LIN {X 0,Y 509.862,Z 318.469,A -85,B 0,C 180,E1 -5560.681,E2 -5560.681} C_VEL
LIN {X 0,Y 509.875,Z 318.471,A -85,B 0,C 180,E1 -5563.174,E2 -5563.174} C_VEL
LIN {X 0,Y 509.873,Z 318.475,A -85,B 0,C 180,E1 -5565.634,E2 -5565.634} C_VEL
LIN {X 0,Y 509.913,Z 318.465,A -85,B 0,C 180,E1 -5568.874,E2 -5568.874} C_VEL
LIN {X 0,Y 509.951,Z 318.459,A -85,B 0,C 180,E1 -5572.078,E2 -5572.078} C_VEL
LIN {X 0,Y 509.98,Z 318.455,A -85,B 0,C 180,E1 -5574.464,E2 -5574.464} C_VEL
LIN {X 0,Y 510.056,Z 318.449,A -85,B 0,C 180,E1 -5577.63,E2 -5577.63} C_VEL
LIN {X 0,Y 510.062,Z 318.448,A -85,B 0,C 180,E1 -5580.789,E2 -5580.789} C_VEL
LIN {X 0,Y 509.954,Z 318.466,A -85,B 0,C 180,E1 -5583.16,E2 -5583.16} C_VEL
LIN {X 0,Y 509.953,Z 318.459,A -85,B 0,C 180,E1 -5586.329,E2 -5586.329} C_VEL
LIN {X 0,Y 509.913,Z 318.468,A -85,B 0,C 180,E1 -5588.72,E2 -5588.72} C_VEL
LIN {X 0,Y 509.903,Z 318.464,A -85,B 0,C 180,E1 -5591.931,E2 -5591.931} C_VEL
LIN {X 0,Y 509.892,Z 318.469,A -85,B 0,C 180,E1 -5595.241,E2 -5595.241} C_VEL
LIN {X 0,Y 509.887,Z 318.467,A -85,B 0,C 180,E1 -5598.001,E2 -5598.001} C_VEL
LIN {X 0,Y 509.848,Z 318.475,A -85,B 0,C 180,E1 -5601.001,E2 -5601.001} C_VEL
LIN {X 0,Y 509.862,Z 318.476,A -85,B 0,C 180,E1 -5604.426,E2 -5604.426} C_VEL
LIN {X 0,Y 509.882,Z 318.469,A -85,B 0,C 180,E1 -5607.055,E2 -5607.055} C_VEL
LIN {X 0,Y 509.854,Z 318.471,A -85,B 0,C 180,E1 -5609.751,E2 -5609.751} C_VEL
LIN {X 0,Y 509.874,Z 318.471,A -85,B 0,C 180,E1 -5612.774,E2 -5612.774} C_VEL
LIN {X 0,Y 509.836,Z 318.473,A -85,B 0,C 180,E1 -5615.58,E2 -5615.58} C_VEL
LIN {X 0,Y 509.849,Z 318.479,A -85,B 0,C 180,E1 -5618.337,E2 -5618.337} C_VEL
LIN {X 0,Y 509.862,Z 318.47,A -85,B 0,C 180,E1 -5621.424,E2 -5621.424} C_VEL
LIN {X 0,Y 509.853,Z 318.472,A -85,B 0,C 180,E1 -5624.668,E2 -5624.668} C_VEL
LIN {X 0,Y 509.858,Z 318.478,A -85,B 0,C 180,E1 -5628.102,E2 -5628.102} C_VEL
LIN {X 0,Y 509.857,Z 318.471,A -85,B 0,C 180,E1 -5630.649,E2 -5630.649} C_VEL
LIN {X 0,Y 509.827,Z 318.478,A -85,B 0,C 180,E1 -5633.723,E2 -5633.723} C_VEL
LIN {X 0,Y 509.159,Z 318.56,A -85,B 0,C 180,E1 -5634.382,E2 -5634.382} C_VEL
LIN {X 0,Y 506.343,Z 318.911,A -85,B 0,C 180,E1 -5635.454,E2 -5635.454} C_VEL
LIN {X 0,Y 503.953,Z 319.208,A -85,B 0,C 180,E1 -5636.318,E2 -5636.318} C_VEL
LIN {X 0,Y 502.905,Z 319.336,A -85,B 0,C 180,E1 -5636.984,E2 -5636.984} C_VEL
LIN {X 0,Y 502.807,Z 319.349,A -85,B 0,C 180,E1 -5637.21,E2 -5637.21} C_VEL
LIN {X 0,Y 502.811,Z 319.352,A -85,B 0,C 180,E1 -5640.065,E2 -5640.065} C_VEL
LIN {X 0,Y 502.832,Z 319.345,A -85,B 0,C 180,E1 -5642.533,E2 -5642.533} C_VEL
LIN {X 0,Y 502.823,Z 319.351,A -85,B 0,C 180,E1 -5645.299,E2 -5645.299} C_VEL
LIN {X 0,Y 502.776,Z 319.357,A -85,B 0,C 180,E1 -5647.826,E2 -5647.826} C_VEL
LIN {X 0,Y 502.822,Z 319.346,A -85,B 0,C 180,E1 -5650.4,E2 -5650.4} C_VEL
LIN {X 0,Y 502.831,Z 319.35,A -85,B 0,C 180,E1 -5652.932,E2 -5652.932} C_VEL
LIN {X 0,Y 502.848,Z 319.352,A -85,B 0,C 180,E1 -5655.429,E2 -5655.429} C_VEL
LIN {X 0,Y 502.874,Z 319.343,A -85,B 0,C 180,E1 -5658.717,E2 -5658.717} C_VEL
LIN {X 0,Y 502.899,Z 319.34,A -85,B 0,C 180,E1 -5661.967,E2 -5661.967} C_VEL
LIN {X 0,Y 502.939,Z 319.335,A -85,B 0,C 180,E1 -5664.387,E2 -5664.387} C_VEL
LIN {X 0,Y 503.023,Z 319.325,A -85,B 0,C 180,E1 -5667.598,E2 -5667.598} C_VEL
LIN {X 0,Y 503.025,Z 319.324,A -85,B 0,C 180,E1 -5670,E2 -5670} C_VEL
LIN {X 0,Y 503.023,Z 319.325,A -85,B 0,C 180,E1 -5672.402,E2 -5672.402} C_VEL
LIN {X 0,Y 502.939,Z 319.335,A -85,B 0,C 180,E1 -5675.613,E2 -5675.613} C_VEL
LIN {X 0,Y 502.899,Z 319.34,A -85,B 0,C 180,E1 -5678.033,E2 -5678.033} C_VEL
LIN {X 0,Y 502.874,Z 319.343,A -85,B 0,C 180,E1 -5681.283,E2 -5681.283} C_VEL
LIN {X 0,Y 502.848,Z 319.352,A -85,B 0,C 180,E1 -5684.571,E2 -5684.571} C_VEL
LIN {X 0,Y 502.859,Z 319.345,A -85,B 0,C 180,E1 -5687.907,E2 -5687.907} C_VEL
LIN {X 0,Y 502.825,Z 319.354,A -85,B 0,C 180,E1 -5690.536,E2 -5690.536} C_VEL
LIN {X 0,Y 502.788,Z 319.352,A -85,B 0,C 180,E1 -5693.041,E2 -5693.041} C_VEL
LIN {X 0,Y 502.838,Z 319.345,A -85,B 0,C 180,E1 -5695.676,E2 -5695.676} C_VEL
LIN {X 0,Y 502.837,Z 319.353,A -85,B 0,C 180,E1 -5698.373,E2 -5698.373} C_VEL
LIN {X 0,Y 502.793,Z 319.351,A -85,B 0,C 180,E1 -5701.5,E2 -5701.5} C_VEL
LIN {X 0,Y 502.801,Z 319.354,A -85,B 0,C 180,E1 -5704.444,E2 -5704.444} C_VEL
LIN {X 0,Y 502.777,Z 319.352,A -85,B 0,C 180,E1 -5707.178,E2 -5707.178} C_VEL
LIN {X 0,Y 502.818,Z 319.356,A -85,B 0,C 180,E1 -5710.012,E2 -5710.012} C_VEL
LIN {X 0,Y 502.77,Z 319.354,A -85,B 0,C 180,E1 -5713.231,E2 -5713.231} C_VEL
LIN {X 0,Y 502.787,Z 319.356,A -85,B 0,C 180,E1 -5715.662,E2 -5715.662} C_VEL
LIN {X 0,Y 502.832,Z 319.354,A -85,B 0,C 180,E1 -5717.865,E2 -5717.865} C_VEL
LIN {X 0,Y 502.807,Z 319.349,A -85,B 0,C 180,E1 -5721.025,E2 -5721.025} C_VEL
LIN {X 0,Y 502.771,Z 319.355,A -85,B 0,C 180,E1 -5724.169,E2 -5724.169} C_VEL
LIN {X 0,Y 502.83,Z 319.347,A -85,B 0,C 180,E1 -5726.994,E2 -5726.994} C_VEL
LIN {X 0,Y 502.812,Z 319.35,A -85,B 0,C 180,E1 -5730.065,E2 -5730.065} C_VEL
LIN {X 0,Y 502.831,Z 319.345,A -85,B 0,C 180,E1 -5732.534,E2 -5732.534} C_VEL
LIN {X 0,Y 502.824,Z 319.353,A -85,B 0,C 180,E1 -5735.299,E2 -5735.299} C_VEL
LIN {X 0,Y 502.778,Z 319.354,A -85,B 0,C 180,E1 -5737.827,E2 -5737.827} C_VEL
LIN {X 0,Y 502.823,Z 319.346,A -85,B 0,C 180,E1 -5740.401,E2 -5740.401} C_VEL
LIN {X 0,Y 502.832,Z 319.35,A -85,B 0,C 180,E1 -5742.932,E2 -5742.932} C_VEL
LIN {X 0,Y 502.843,Z 319.349,A -85,B 0,C 180,E1 -5745.43,E2 -5745.43} C_VEL
LIN {X 0,Y 502.876,Z 319.343,A -85,B 0,C 180,E1 -5748.717,E2 -5748.717} C_VEL
LIN {X 0,Y 502.9,Z 319.337,A -85,B 0,C 180,E1 -5751.967,E2 -5751.967} C_VEL
LIN {X 0,Y 502.933,Z 319.334,A -85,B 0,C 180,E1 -5754.387,E2 -5754.387} C_VEL
LIN {X 0,Y 503.024,Z 319.322,A -85,B 0,C 180,E1 -5757.598,E2 -5757.598} C_VEL
LIN {X 0,Y 503.034,Z 319.329,A -85,B 0,C 180,E1 -5760.801,E2 -5760.801} C_VEL
LIN {X 0,Y 502.896,Z 319.34,A -85,B 0,C 180,E1 -5763.205,E2 -5763.205} C_VEL
LIN {X 0,Y 502.906,Z 319.341,A -85,B 0,C 180,E1 -5766.419,E2 -5766.419} C_VEL
LIN {X 0,Y 502.874,Z 319.345,A -85,B 0,C 180,E1 -5768.844,E2 -5768.844} C_VEL
LIN {X 0,Y 502.846,Z 319.346,A -85,B 0,C 180,E1 -5772.102,E2 -5772.102} C_VEL
LIN {X 0,Y 502.849,Z 319.343,A -85,B 0,C 180,E1 -5775.4,E2 -5775.4} C_VEL
LIN {X 0,Y 502.826,Z 319.349,A -85,B 0,C 180,E1 -5778.752,E2 -5778.752} C_VEL
LIN {X 0,Y 502.783,Z 319.351,A -85,B 0,C 180,E1 -5781.312,E2 -5781.312} C_VEL
LIN {X 0,Y 502.776,Z 319.356,A -85,B 0,C 180,E1 -5783.915,E2 -5783.915} C_VEL
LIN {X 0,Y 502.865,Z 319.344,A -85,B 0,C 180,E1 -5786.566,E2 -5786.566} C_VEL
LIN {X 0,Y 502.824,Z 319.346,A -85,B 0,C 180,E1 -5789.288,E2 -5789.288} C_VEL
LIN {X 0,Y 502.784,Z 319.36,A -85,B 0,C 180,E1 -5792.085,E2 -5792.085} C_VEL
LIN {X 0,Y 502.799,Z 319.349,A -85,B 0,C 180,E1 -5794.966,E2 -5794.966} C_VEL
LIN {X 0,Y 502.794,Z 319.359,A -85,B 0,C 180,E1 -5797.954,E2 -5797.954} C_VEL
LIN {X 0,Y 502.821,Z 319.352,A -85,B 0,C 180,E1 -5801.066,E2 -5801.066} C_VEL
LIN {X 0,Y 502.792,Z 319.531,A -85,B 0,C 180,E1 -5803.377,E2 -5803.377} C_VEL
LIN {X 0,Y 503.366,Z 323.551,A -85,B 0,C 180,E1 -5806.555,E2 -5806.555} C_VEL
LIN {X 0,Y 503.464,Z 326.838,A -85,B 0,C 180,E1 -5808.921,E2 -5808.921} C_VEL
LIN {X 0,Y 503.339,Z 331.622,A -85,B 0,C 180,E1 -5812.095,E2 -5812.095} C_VEL
LIN {X 0,Y 503.119,Z 336.421,A -85,B 0,C 180,E1 -5815.06,E2 -5815.06} C_VEL
LIN {X 0,Y 502.955,Z 341.324,A -85,B 0,C 180,E1 -5817.928,E2 -5817.928} C_VEL
LIN {X 0,Y 502.767,Z 346.348,A -85,B 0,C 180,E1 -5820.709,E2 -5820.709} C_VEL
LIN {X 0,Y 502.617,Z 351.579,A -85,B 0,C 180,E1 -5823.496,E2 -5823.496} C_VEL
LIN {X 0,Y 502.426,Z 356.59,A -85,B 0,C 180,E1 -5826.068,E2 -5826.068} C_VEL
LIN {X 0,Y 502.342,Z 361.823,A -85,B 0,C 180,E1 -5828.669,E2 -5828.669} C_VEL
LIN {X 0,Y 502.248,Z 367.111,A -85,B 0,C 180,E1 -5831.226,E2 -5831.226} C_VEL
LIN {X 0,Y 502.175,Z 372.422,A -85,B 0,C 180,E1 -5833.746,E2 -5833.746} C_VEL
LIN {X 0,Y 502.176,Z 376.661,A -85,B 0,C 180,E1 -5835.72,E2 -5835.72} C_VEL
LIN {X 0,Y 504.336,Z 390.065,A -85,B 0,C 180,E1 -5836.133,E2 -5836.133} C_VEL
LIN {X 0,Y 504.45,Z 397.294,A -85,B 0,C 180,E1 -5836.402,E2 -5836.402} C_VEL
LIN {X 0,Y 504.208,Z 406.373,A -85,B 0,C 180,E1 -5836.806,E2 -5836.806} C_VEL
LIN {X 0,Y 503.872,Z 416.43,A -85,B 0,C 180,E1 -5837.368,E2 -5837.368} C_VEL
LIN {X 0,Y 503.598,Z 424.509,A -85,B 0,C 180,E1 -5837.917,E2 -5837.917} C_VEL
LIN {X 0,Y 503.364,Z 433.242,A -85,B 0,C 180,E1 -5838.626,E2 -5838.626} C_VEL
LIN {X 0,Y 503.096,Z 440.64,A -85,B 0,C 180,E1 -5839.333,E2 -5839.333} C_VEL
LIN {X 0,Y 502.873,Z 447.862,A -85,B 0,C 180,E1 -5840.142,E2 -5840.142} C_VEL
LIN {X 0,Y 502.658,Z 454.064,A -85,B 0,C 180,E1 -5840.95,E2 -5840.95} C_VEL
LIN {X 0,Y 502.487,Z 460.603,A -85,B 0,C 180,E1 -5841.96,E2 -5841.96} C_VEL
LIN {X 0,Y 502.332,Z 466.157,A -85,B 0,C 180,E1 -5842.989,E2 -5842.989} C_VEL
LIN {X 0,Y 502.233,Z 470.593,A -85,B 0,C 180,E1 -5843.976,E2 -5843.976} C_VEL
LIN {X 0,Y 502.115,Z 474.913,A -85,B 0,C 180,E1 -5845.183,E2 -5845.183} C_VEL
LIN {X 0,Y 502.14,Z 477.278,A -85,B 0,C 180,E1 -5845.987,E2 -5845.987} C_VEL
LIN {X 0,Y 502.121,Z 479.073,A -85,B 0,C 180,E1 -5846.791,E2 -5846.791} C_VEL
LIN {X 0,Y 502.037,Z 481.512,A -85,B 0,C 180,E1 -5848.396,E2 -5848.396} C_VEL
LIN {X 0,Y 501.99,Z 482.097,A -85,B 0,C 180,E1 -5849.198,E2 -5849.198} C_VEL
LIN {X 0,Y 501.99,Z 482.097,A -85,B 0,C 180,E1 -5850.802,E2 -5850.802} C_VEL
LIN {X 0,Y 502.037,Z 481.512,A -85,B 0,C 180,E1 -5851.604,E2 -5851.604} C_VEL
LIN {X 0,Y 502.121,Z 479.073,A -85,B 0,C 180,E1 -5853.209,E2 -5853.209} C_VEL
LIN {X 0,Y 502.107,Z 476.128,A -85,B 0,C 180,E1 -5854.415,E2 -5854.415} C_VEL
LIN {X 0,Y 502.217,Z 472.146,A -85,B 0,C 180,E1 -5855.622,E2 -5855.622} C_VEL
LIN {X 0,Y 502.277,Z 467.21,A -85,B 0,C 180,E1 -5856.79,E2 -5856.79} C_VEL
LIN {X 0,Y 502.418,Z 461.757,A -85,B 0,C 180,E1 -5857.839,E2 -5857.839} C_VEL
LIN {X 0,Y 502.611,Z 455.441,A -85,B 0,C 180,E1 -5858.848,E2 -5858.848} C_VEL
LIN {X 0,Y 502.826,Z 449.489,A -85,B 0,C 180,E1 -5859.655,E2 -5859.655} C_VEL
LIN {X 0,Y 503.01,Z 442.559,A -85,B 0,C 180,E1 -5860.465,E2 -5860.465} C_VEL
LIN {X 0,Y 503.324,Z 434.377,A -85,B 0,C 180,E1 -5861.273,E2 -5861.273} C_VEL
LIN {X 0,Y 503.624,Z 425.863,A -85,B 0,C 180,E1 -5861.98,E2 -5861.98} C_VEL
LIN {X 0,Y 503.807,Z 417.91,A -85,B 0,C 180,E1 -5862.541,E2 -5862.541} C_VEL
LIN {X 0,Y 504.092,Z 408.386,A -85,B 0,C 180,E1 -5863.094,E2 -5863.094} C_VEL
LIN {X 0,Y 504.404,Z 398.582,A -85,B 0,C 180,E1 -5863.548,E2 -5863.548} C_VEL
LIN {X 0,Y 504.443,Z 390.833,A -85,B 0,C 180,E1 -5863.842,E2 -5863.842} C_VEL
LIN {X 0,Y 502.465,Z 378.896,A -85,B 0,C 180,E1 -5864.217,E2 -5864.217} C_VEL
LIN {X 0,Y 502.167,Z 376.661,A -85,B 0,C 180,E1 -5864.28,E2 -5864.28} C_VEL
LIN {X 0,Y 502.212,Z 370.632,A -85,B 0,C 180,E1 -5867.09,E2 -5867.09} C_VEL
LIN {X 0,Y 502.34,Z 363.567,A -85,B 0,C 180,E1 -5870.473,E2 -5870.473} C_VEL
LIN {X 0,Y 502.406,Z 358.325,A -85,B 0,C 180,E1 -5873.059,E2 -5873.059} C_VEL
LIN {X 0,Y 502.533,Z 353.134,A -85,B 0,C 180,E1 -5875.692,E2 -5875.692} C_VEL
LIN {X 0,Y 502.692,Z 347.991,A -85,B 0,C 180,E1 -5878.382,E2 -5878.382} C_VEL
LIN {X 0,Y 502.89,Z 342.977,A -85,B 0,C 180,E1 -5881.137,E2 -5881.137} C_VEL
LIN {X 0,Y 503.066,Z 338.021,A -85,B 0,C 180,E1 -5883.974,E2 -5883.974} C_VEL
LIN {X 0,Y 503.247,Z 333.191,A -85,B 0,C 180,E1 -5886.906,E2 -5886.906} C_VEL
LIN {X 0,Y 503.406,Z 328.47,A -85,B 0,C 180,E1 -5889.956,E2 -5889.956} C_VEL
LIN {X 0,Y 503.471,Z 325.105,A -85,B 0,C 180,E1 -5892.282,E2 -5892.282} C_VEL
LIN {X 0,Y 503.174,Z 322.074,A -85,B 0,C 180,E1 -5894.574,E2 -5894.574} C_VEL
LIN {X 0,Y 502.774,Z 319.359,A -85,B 0,C 180,E1 -5896.768,E2 -5896.768} C_VEL
LIN {X 0,Y 502.819,Z 319.352,A -85,B 0,C 180,E1 -5899.005,E2 -5899.005} C_VEL
LIN {X 0,Y 502.794,Z 319.359,A -85,B 0,C 180,E1 -5902.046,E2 -5902.046} C_VEL
LIN {X 0,Y 502.799,Z 319.352,A -85,B 0,C 180,E1 -5905.034,E2 -5905.034} C_VEL
LIN {X 0,Y 502.784,Z 319.36,A -85,B 0,C 180,E1 -5907.915,E2 -5907.915} C_VEL
LIN {X 0,Y 502.824,Z 319.346,A -85,B 0,C 180,E1 -5910.712,E2 -5910.712} C_VEL
LIN {X 0,Y 502.863,Z 319.345,A -85,B 0,C 180,E1 -5913.439,E2 -5913.439} C_VEL
LIN {X 0,Y 502.776,Z 319.356,A -85,B 0,C 180,E1 -5916.085,E2 -5916.085} C_VEL
LIN {X 0,Y 502.783,Z 319.351,A -85,B 0,C 180,E1 -5918.688,E2 -5918.688} C_VEL
LIN {X 0,Y 502.826,Z 319.349,A -85,B 0,C 180,E1 -5921.248,E2 -5921.248} C_VEL
LIN {X 0,Y 502.849,Z 319.343,A -85,B 0,C 180,E1 -5924.6,E2 -5924.6} C_VEL
LIN {X 0,Y 502.876,Z 319.341,A -85,B 0,C 180,E1 -5928.039,E2 -5928.039} C_VEL
LIN {X 0,Y 502.874,Z 319.345,A -85,B 0,C 180,E1 -5931.156,E2 -5931.156} C_VEL
LIN {X 0,Y 502.906,Z 319.341,A -85,B 0,C 180,E1 -5933.581,E2 -5933.581} C_VEL
LIN {X 0,Y 502.896,Z 319.34,A -85,B 0,C 180,E1 -5936.795,E2 -5936.795} C_VEL
LIN {X 0,Y 503.034,Z 319.329,A -85,B 0,C 180,E1 -5939.199,E2 -5939.199} C_VEL
LIN {X 0,Y 503.024,Z 319.322,A -85,B 0,C 180,E1 -5942.402,E2 -5942.402} C_VEL
LIN {X 0,Y 502.933,Z 319.334,A -85,B 0,C 180,E1 -5945.613,E2 -5945.613} C_VEL
LIN {X 0,Y 502.9,Z 319.337,A -85,B 0,C 180,E1 -5948.033,E2 -5948.033} C_VEL
LIN {X 0,Y 502.876,Z 319.343,A -85,B 0,C 180,E1 -5951.283,E2 -5951.283} C_VEL
LIN {X 0,Y 502.843,Z 319.349,A -85,B 0,C 180,E1 -5954.57,E2 -5954.57} C_VEL
LIN {X 0,Y 502.86,Z 319.342,A -85,B 0,C 180,E1 -5957.907,E2 -5957.907} C_VEL
LIN {X 0,Y 502.826,Z 319.352,A -85,B 0,C 180,E1 -5960.536,E2 -5960.536} C_VEL
LIN {X 0,Y 502.789,Z 319.354,A -85,B 0,C 180,E1 -5963.04,E2 -5963.04} C_VEL
LIN {X 0,Y 502.837,Z 319.345,A -85,B 0,C 180,E1 -5965.675,E2 -5965.675} C_VEL
LIN {X 0,Y 502.837,Z 319.352,A -85,B 0,C 180,E1 -5968.372,E2 -5968.372} C_VEL
LIN {X 0,Y 502.793,Z 319.35,A -85,B 0,C 180,E1 -5971.499,E2 -5971.499} C_VEL
LIN {X 0,Y 502.801,Z 319.356,A -85,B 0,C 180,E1 -5974.444,E2 -5974.444} C_VEL
LIN {X 0,Y 502.777,Z 319.352,A -85,B 0,C 180,E1 -5977.178,E2 -5977.178} C_VEL
LIN {X 0,Y 502.819,Z 319.353,A -85,B 0,C 180,E1 -5980.012,E2 -5980.012} C_VEL
LIN {X 0,Y 502.82,Z 319.355,A -85,B 0,C 180,E1 -5982.202,E2 -5982.202} C_VEL
LIN {X 0,Y 502.797,Z 319.351,A -85,B 0,C 180,E1 -5985.468,E2 -5985.468} C_VEL
LIN {X 0,Y 502.823,Z 319.346,A -85,B 0,C 180,E1 -5989.004,E2 -5989.004} C_VEL
LIN {X 0,Y 502.791,Z 319.357,A -85,B 0,C 180,E1 -5992.046,E2 -5992.046} C_VEL
LIN {X 0,Y 502.804,Z 319.349,A -85,B 0,C 180,E1 -5995.035,E2 -5995.035} C_VEL
LIN {X 0,Y 502.807,Z 319.349,A -85,B 0,C 180,E1 -5997.21,E2 -5997.21} C_VEL
LIN {X 0,Y 502.106,Z 319.443,A -85,B 0,C 180,E1 -5997.878,E2 -5997.878} C_VEL
LIN {X 0,Y 499.241,Z 319.794,A -85,B 0,C 180,E1 -5998.964,E2 -5998.964} C_VEL
LIN {X 0,Y 496.845,Z 320.098,A -85,B 0,C 180,E1 -5999.839,E2 -5999.839} C_VEL
LIN {X 0,Y 495.828,Z 320.219,A -85,B 0,C 180,E1 -6000.515,E2 -6000.515} C_VEL
LIN {X 0,Y 495.749,Z 320.227,A -85,B 0,C 180,E1 -6000.743,E2 -6000.743} C_VEL
LIN {X 0,Y 495.796,Z 320.226,A -85,B 0,C 180,E1 -6003.933,E2 -6003.933} C_VEL
LIN {X 0,Y 495.756,Z 320.23,A -85,B 0,C 180,E1 -6007.139,E2 -6007.139} C_VEL
LIN {X 0,Y 495.774,Z 320.226,A -85,B 0,C 180,E1 -6010.11,E2 -6010.11} C_VEL
LIN {X 0,Y 495.783,Z 320.226,A -85,B 0,C 180,E1 -6012.681,E2 -6012.681} C_VEL
LIN {X 0,Y 495.791,Z 320.23,A -85,B 0,C 180,E1 -6015.217,E2 -6015.217} C_VEL
LIN {X 0,Y 495.849,Z 320.218,A -85,B 0,C 180,E1 -6018.555,E2 -6018.555} C_VEL
LIN {X 0,Y 495.87,Z 320.216,A -85,B 0,C 180,E1 -6021.852,E2 -6021.852} C_VEL
LIN {X 0,Y 495.896,Z 320.212,A -85,B 0,C 180,E1 -6024.307,E2 -6024.307} C_VEL
LIN {X 0,Y 495.992,Z 320.202,A -85,B 0,C 180,E1 -6027.564,E2 -6027.564} C_VEL
LIN {X 0,Y 495.996,Z 320.2,A -85,B 0,C 180,E1 -6030,E2 -6030} C_VEL
LIN {X 0,Y 495.992,Z 320.202,A -85,B 0,C 180,E1 -6032.436,E2 -6032.436} C_VEL
LIN {X 0,Y 495.896,Z 320.212,A -85,B 0,C 180,E1 -6035.693,E2 -6035.693} C_VEL
LIN {X 0,Y 495.87,Z 320.216,A -85,B 0,C 180,E1 -6038.148,E2 -6038.148} C_VEL
LIN {X 0,Y 495.849,Z 320.218,A -85,B 0,C 180,E1 -6041.445,E2 -6041.445} C_VEL
LIN {X 0,Y 495.791,Z 320.23,A -85,B 0,C 180,E1 -6044.783,E2 -6044.783} C_VEL
LIN {X 0,Y 495.795,Z 320.227,A -85,B 0,C 180,E1 -6048.171,E2 -6048.171} C_VEL
LIN {X 0,Y 495.77,Z 320.23,A -85,B 0,C 180,E1 -6050.756,E2 -6050.756} C_VEL
LIN {X 0,Y 495.744,Z 320.228,A -85,B 0,C 180,E1 -6053.387,E2 -6053.387} C_VEL
LIN {X 0,Y 495.796,Z 320.226,A -85,B 0,C 180,E1 -6056.067,E2 -6056.067} C_VEL
LIN {X 0,Y 495.769,Z 320.227,A -85,B 0,C 180,E1 -6058.815,E2 -6058.815} C_VEL
LIN {X 0,Y 495.755,Z 320.229,A -85,B 0,C 180,E1 -6061.726,E2 -6061.726} C_VEL
LIN {X 0,Y 495.771,Z 320.227,A -85,B 0,C 180,E1 -6064.695,E2 -6064.695} C_VEL
LIN {X 0,Y 495.728,Z 320.232,A -85,B 0,C 180,E1 -6067.562,E2 -6067.562} C_VEL
LIN {X 0,Y 495.776,Z 320.225,A -85,B 0,C 180,E1 -6070.699,E2 -6070.699} C_VEL
LIN {X 0,Y 495.73,Z 320.238,A -85,B 0,C 180,E1 -6074.001,E2 -6074.001} C_VEL
LIN {X 0,Y 495.759,Z 320.227,A -85,B 0,C 180,E1 -6077.121,E2 -6077.121} C_VEL
LIN {X 0,Y 495.78,Z 320.225,A -85,B 0,C 180,E1 -6080.365,E2 -6080.365} C_VEL
LIN {X 0,Y 495.724,Z 320.236,A -85,B 0,C 180,E1 -6083.456,E2 -6083.456} C_VEL
LIN {X 0,Y 495.756,Z 320.227,A -85,B 0,C 180,E1 -6086.436,E2 -6086.436} C_VEL
LIN {X 0,Y 495.75,Z 320.232,A -85,B 0,C 180,E1 -6089.313,E2 -6089.313} C_VEL
LIN {X 0,Y 495.778,Z 320.225,A -85,B 0,C 180,E1 -6092.109,E2 -6092.109} C_VEL
LIN {X 0,Y 495.785,Z 320.224,A -85,B 0,C 180,E1 -6094.833,E2 -6094.833} C_VEL
LIN {X 0,Y 495.746,Z 320.235,A -85,B 0,C 180,E1 -6097.495,E2 -6097.495} C_VEL
LIN {X 0,Y 495.775,Z 320.225,A -85,B 0,C 180,E1 -6100.11,E2 -6100.11} C_VEL
LIN {X 0,Y 495.784,Z 320.225,A -85,B 0,C 180,E1 -6102.682,E2 -6102.682} C_VEL
LIN {X 0,Y 495.788,Z 320.231,A -85,B 0,C 180,E1 -6105.218,E2 -6105.218} C_VEL
LIN {X 0,Y 495.85,Z 320.217,A -85,B 0,C 180,E1 -6108.555,E2 -6108.555} C_VEL
LIN {X 0,Y 495.871,Z 320.212,A -85,B 0,C 180,E1 -6111.852,E2 -6111.852} C_VEL
LIN {X 0,Y 495.889,Z 320.211,A -85,B 0,C 180,E1 -6114.307,E2 -6114.307} C_VEL
LIN {X 0,Y 495.993,Z 320.198,A -85,B 0,C 180,E1 -6117.564,E2 -6117.564} C_VEL
LIN {X 0,Y 496.004,Z 320.204,A -85,B 0,C 180,E1 -6120.812,E2 -6120.812} C_VEL
LIN {X 0,Y 495.84,Z 320.218,A -85,B 0,C 180,E1 -6123.251,E2 -6123.251} C_VEL
LIN {X 0,Y 495.861,Z 320.22,A -85,B 0,C 180,E1 -6126.511,E2 -6126.511} C_VEL
LIN {X 0,Y 495.842,Z 320.219,A -85,B 0,C 180,E1 -6128.97,E2 -6128.97} C_VEL
LIN {X 0,Y 495.828,Z 320.22,A -85,B 0,C 180,E1 -6132.035,E2 -6132.035} C_VEL
LIN {X 0,Y 495.824,Z 320.218,A -85,B 0,C 180,E1 -6135.452,E2 -6135.452} C_VEL
LIN {X 0,Y 495.779,Z 320.23,A -85,B 0,C 180,E1 -6138.238,E2 -6138.238} C_VEL
LIN {X 0,Y 495.774,Z 320.227,A -85,B 0,C 180,E1 -6140.757,E2 -6140.757} C_VEL
LIN {X 0,Y 495.743,Z 320.228,A -85,B 0,C 180,E1 -6143.388,E2 -6143.388} C_VEL
LIN {X 0,Y 495.824,Z 320.22,A -85,B 0,C 180,E1 -6146.75,E2 -6146.75} C_VEL
LIN {X 0,Y 495.767,Z 320.229,A -85,B 0,C 180,E1 -6149.747,E2 -6149.747} C_VEL
LIN {X 0,Y 495.768,Z 320.227,A -85,B 0,C 180,E1 -6152.595,E2 -6152.595} C_VEL
LIN {X 0,Y 495.749,Z 320.231,A -85,B 0,C 180,E1 -6155.538,E2 -6155.538} C_VEL
LIN {X 0,Y 495.765,Z 320.23,A -85,B 0,C 180,E1 -6158.769,E2 -6158.769} C_VEL
LIN {X 0,Y 495.757,Z 320.235,A -85,B 0,C 180,E1 -6161.782,E2 -6161.782} C_VEL
LIN {X 0,Y 495.727,Z 320.238,A -85,B 0,C 180,E1 -6162.883,E2 -6162.883} C_VEL
LIN {X 0,Y 496.278,Z 324.069,A -85,B 0,C 180,E1 -6166.06,E2 -6166.06} C_VEL
LIN {X 0,Y 496.48,Z 327.071,A -85,B 0,C 180,E1 -6168.294,E2 -6168.294} C_VEL
LIN {X 0,Y 496.336,Z 331.702,A -85,B 0,C 180,E1 -6171.463,E2 -6171.463} C_VEL
LIN {X 0,Y 496.19,Z 335.407,A -85,B 0,C 180,E1 -6173.838,E2 -6173.838} C_VEL
LIN {X 0,Y 495.998,Z 340.155,A -85,B 0,C 180,E1 -6176.72,E2 -6176.72} C_VEL
LIN {X 0,Y 495.782,Z 345.607,A -85,B 0,C 180,E1 -6179.85,E2 -6179.85} C_VEL
LIN {X 0,Y 495.565,Z 351.404,A -85,B 0,C 180,E1 -6183.011,E2 -6183.011} C_VEL
LIN {X 0,Y 495.383,Z 356.535,A -85,B 0,C 180,E1 -6185.706,E2 -6185.706} C_VEL
LIN {X 0,Y 495.286,Z 361.727,A -85,B 0,C 180,E1 -6188.35,E2 -6188.35} C_VEL
LIN {X 0,Y 495.174,Z 366.998,A -85,B 0,C 180,E1 -6190.947,E2 -6190.947} C_VEL
LIN {X 0,Y 495.097,Z 372.288,A -85,B 0,C 180,E1 -6193.507,E2 -6193.507} C_VEL
LIN {X 0,Y 495.067,Z 376.529,A -85,B 0,C 180,E1 -6195.524,E2 -6195.524} C_VEL
LIN {X 0,Y 496.754,Z 387.005,A -85,B 0,C 180,E1 -6195.832,E2 -6195.832} C_VEL
LIN {X 0,Y 497.611,Z 393.233,A -85,B 0,C 180,E1 -6196.056,E2 -6196.056} C_VEL
LIN {X 0,Y 497.318,Z 404.161,A -85,B 0,C 180,E1 -6196.516,E2 -6196.516} C_VEL
LIN {X 0,Y 496.991,Z 415.121,A -85,B 0,C 180,E1 -6197.119,E2 -6197.119} C_VEL
LIN {X 0,Y 496.628,Z 424.312,A -85,B 0,C 180,E1 -6197.745,E2 -6197.745} C_VEL
LIN {X 0,Y 496.383,Z 433.046,A -85,B 0,C 180,E1 -6198.464,E2 -6198.464} C_VEL
LIN {X 0,Y 496.104,Z 440.443,A -85,B 0,C 180,E1 -6199.181,E2 -6199.181} C_VEL
LIN {X 0,Y 495.856,Z 447.665,A -85,B 0,C 180,E1 -6200.001,E2 -6200.001} C_VEL
LIN {X 0,Y 495.624,Z 453.868,A -85,B 0,C 180,E1 -6200.821,E2 -6200.821} C_VEL
LIN {X 0,Y 495.416,Z 460.406,A -85,B 0,C 180,E1 -6201.845,E2 -6201.845} C_VEL
LIN {X 0,Y 495.273,Z 464.907,A -85,B 0,C 180,E1 -6202.663,E2 -6202.663} C_VEL
LIN {X 0,Y 495.135,Z 469.869,A -85,B 0,C 180,E1 -6203.75,E2 -6203.75} C_VEL
LIN {X 0,Y 495.111,Z 473.479,A -85,B 0,C 180,E1 -6204.706,E2 -6204.706} C_VEL
LIN {X 0,Y 495.034,Z 477.081,A -85,B 0,C 180,E1 -6205.929,E2 -6205.929} C_VEL
LIN {X 0,Y 495.042,Z 478.878,A -85,B 0,C 180,E1 -6206.745,E2 -6206.745} C_VEL
LIN {X 0,Y 494.963,Z 481.316,A -85,B 0,C 180,E1 -6208.373,E2 -6208.373} C_VEL
LIN {X 0,Y 494.911,Z 481.902,A -85,B 0,C 180,E1 -6209.186,E2 -6209.186} C_VEL
LIN {X 0,Y 494.911,Z 481.902,A -85,B 0,C 180,E1 -6210.814,E2 -6210.814} C_VEL
LIN {X 0,Y 494.963,Z 481.316,A -85,B 0,C 180,E1 -6211.627,E2 -6211.627} C_VEL
LIN {X 0,Y 495.042,Z 478.878,A -85,B 0,C 180,E1 -6213.255,E2 -6213.255} C_VEL
LIN {X 0,Y 495.012,Z 475.932,A -85,B 0,C 180,E1 -6214.479,E2 -6214.479} C_VEL
LIN {X 0,Y 495.136,Z 471.95,A -85,B 0,C 180,E1 -6215.702,E2 -6215.702} C_VEL
LIN {X 0,Y 495.219,Z 466.822,A -85,B 0,C 180,E1 -6216.928,E2 -6216.928} C_VEL
LIN {X 0,Y 495.369,Z 461.561,A -85,B 0,C 180,E1 -6217.951,E2 -6217.951} C_VEL
LIN {X 0,Y 495.573,Z 455.244,A -85,B 0,C 180,E1 -6218.975,E2 -6218.975} C_VEL
LIN {X 0,Y 495.777,Z 449.292,A -85,B 0,C 180,E1 -6219.794,E2 -6219.794} C_VEL
LIN {X 0,Y 496.001,Z 442.362,A -85,B 0,C 180,E1 -6220.615,E2 -6220.615} C_VEL
LIN {X 0,Y 496.328,Z 434.18,A -85,B 0,C 180,E1 -6221.434,E2 -6221.434} C_VEL
LIN {X 0,Y 496.633,Z 425.666,A -85,B 0,C 180,E1 -6222.152,E2 -6222.152} C_VEL
LIN {X 0,Y 496.884,Z 416.714,A -85,B 0,C 180,E1 -6222.782,E2 -6222.782} C_VEL
LIN {X 0,Y 497.186,Z 407.182,A -85,B 0,C 180,E1 -6223.332,E2 -6223.332} C_VEL
LIN {X 0,Y 497.509,Z 398.387,A -85,B 0,C 180,E1 -6223.739,E2 -6223.739} C_VEL
LIN {X 0,Y 497.503,Z 391.482,A -85,B 0,C 180,E1 -6224.013,E2 -6224.013} C_VEL
LIN {X 0,Y 495.404,Z 378.706,A -85,B 0,C 180,E1 -6224.424,E2 -6224.424} C_VEL
LIN {X 0,Y 495.043,Z 376.5,A -85,B 0,C 180,E1 -6224.49,E2 -6224.49} C_VEL
LIN {X 0,Y 495.154,Z 370.498,A -85,B 0,C 180,E1 -6227.341,E2 -6227.341} C_VEL
LIN {X 0,Y 495.255,Z 363.471,A -85,B 0,C 180,E1 -6230.779,E2 -6230.779} C_VEL
LIN {X 0,Y 495.33,Z 358.247,A -85,B 0,C 180,E1 -6233.408,E2 -6233.408} C_VEL
LIN {X 0,Y 495.577,Z 351.933,A -85,B 0,C 180,E1 -6236.692,E2 -6236.692} C_VEL
LIN {X 0,Y 495.749,Z 346.323,A -85,B 0,C 180,E1 -6239.747,E2 -6239.747} C_VEL
LIN {X 0,Y 495.923,Z 341.326,A -85,B 0,C 180,E1 -6242.583,E2 -6242.583} C_VEL
LIN {X 0,Y 496.129,Z 336.46,A -85,B 0,C 180,E1 -6245.506,E2 -6245.506} C_VEL
LIN {X 0,Y 496.299,Z 331.69,A -85,B 0,C 180,E1 -6248.541,E2 -6248.541} C_VEL
LIN {X 0,Y 496.462,Z 327.513,A -85,B 0,C 180,E1 -6251.385,E2 -6251.385} C_VEL
LIN {X 0,Y 496.307,Z 324.284,A -85,B 0,C 180,E1 -6253.764,E2 -6253.764} C_VEL
LIN {X 0,Y 495.85,Z 321.145,A -85,B 0,C 180,E1 -6256.29,E2 -6256.29} C_VEL
LIN {X 0,Y 495.727,Z 320.238,A -85,B 0,C 180,E1 -6257.117,E2 -6257.117} C_VEL
LIN {X 0,Y 495.76,Z 320.234,A -85,B 0,C 180,E1 -6259.953,E2 -6259.953} C_VEL
LIN {X 0,Y 495.729,Z 320.236,A -85,B 0,C 180,E1 -6262.553,E2 -6262.553} C_VEL
LIN {X 0,Y 495.778,Z 320.229,A -85,B 0,C 180,E1 -6265.456,E2 -6265.456} C_VEL
LIN {X 0,Y 495.756,Z 320.23,A -85,B 0,C 180,E1 -6268.363,E2 -6268.363} C_VEL
LIN {X 0,Y 495.788,Z 320.226,A -85,B 0,C 180,E1 -6271.506,E2 -6271.506} C_VEL
LIN {X 0,Y 495.781,Z 320.23,A -85,B 0,C 180,E1 -6273.931,E2 -6273.931} C_VEL
LIN {X 0,Y 495.759,Z 320.228,A -85,B 0,C 180,E1 -6277.139,E2 -6277.139} C_VEL
LIN {X 0,Y 495.771,Z 320.228,A -85,B 0,C 180,E1 -6280.109,E2 -6280.109} C_VEL
LIN {X 0,Y 495.765,Z 320.226,A -85,B 0,C 180,E1 -6282.68,E2 -6282.68} C_VEL
LIN {X 0,Y 495.794,Z 320.226,A -85,B 0,C 180,E1 -6285.217,E2 -6285.217} C_VEL
LIN {X 0,Y 495.851,Z 320.215,A -85,B 0,C 180,E1 -6288.554,E2 -6288.554} C_VEL
LIN {X 0,Y 495.873,Z 320.215,A -85,B 0,C 180,E1 -6291.852,E2 -6291.852} C_VEL
LIN {X 0,Y 495.889,Z 320.21,A -85,B 0,C 180,E1 -6294.306,E2 -6294.306} C_VEL
LIN {X 0,Y 495.993,Z 320.201,A -85,B 0,C 180,E1 -6297.563,E2 -6297.563} C_VEL
LIN {X 0,Y 495.998,Z 320.197,A -85,B 0,C 180,E1 -6300,E2 -6300} C_VEL
LIN {X 0,Y 495.993,Z 320.198,A -85,B 0,C 180,E1 -6302.436,E2 -6302.436} C_VEL
LIN {X 0,Y 495.889,Z 320.211,A -85,B 0,C 180,E1 -6305.693,E2 -6305.693} C_VEL
LIN {X 0,Y 495.871,Z 320.212,A -85,B 0,C 180,E1 -6308.148,E2 -6308.148} C_VEL
LIN {X 0,Y 495.85,Z 320.217,A -85,B 0,C 180,E1 -6311.445,E2 -6311.445} C_VEL
LIN {X 0,Y 495.788,Z 320.231,A -85,B 0,C 180,E1 -6314.782,E2 -6314.782} C_VEL
LIN {X 0,Y 495.784,Z 320.225,A -85,B 0,C 180,E1 -6317.318,E2 -6317.318} C_VEL
LIN {X 0,Y 495.775,Z 320.225,A -85,B 0,C 180,E1 -6319.89,E2 -6319.89} C_VEL
LIN {X 0,Y 495.757,Z 320.232,A -85,B 0,C 180,E1 -6322.86,E2 -6322.86} C_VEL
LIN {X 0,Y 495.788,Z 320.225,A -85,B 0,C 180,E1 -6326.067,E2 -6326.067} C_VEL
LIN {X 0,Y 495.769,Z 320.229,A -85,B 0,C 180,E1 -6328.814,E2 -6328.814} C_VEL
LIN {X 0,Y 495.756,Z 320.228,A -85,B 0,C 180,E1 -6331.726,E2 -6331.726} C_VEL
LIN {X 0,Y 495.771,Z 320.228,A -85,B 0,C 180,E1 -6334.695,E2 -6334.695} C_VEL
LIN {X 0,Y 495.728,Z 320.231,A -85,B 0,C 180,E1 -6337.561,E2 -6337.561} C_VEL
LIN {X 0,Y 495.777,Z 320.226,A -85,B 0,C 180,E1 -6340.698,E2 -6340.698} C_VEL
LIN {X 0,Y 495.731,Z 320.233,A -85,B 0,C 180,E1 -6343.695,E2 -6343.695} C_VEL
LIN {X 0,Y 495.725,Z 320.236,A -85,B 0,C 180,E1 -6346.305,E2 -6346.305} C_VEL
LIN {X 0,Y 495.776,Z 320.225,A -85,B 0,C 180,E1 -6349.301,E2 -6349.301} C_VEL
LIN {X 0,Y 495.728,Z 320.232,A -85,B 0,C 180,E1 -6352.438,E2 -6352.438} C_VEL
LIN {X 0,Y 495.779,Z 320.227,A -85,B 0,C 180,E1 -6355.457,E2 -6355.457} C_VEL
LIN {X 0,Y 495.755,Z 320.228,A -85,B 0,C 180,E1 -6358.364,E2 -6358.364} C_VEL
LIN {X 0,Y 495.749,Z 320.227,A -85,B 0,C 180,E1 -6360.743,E2 -6360.743} C_VEL
LIN {X 0,Y 495.093,Z 320.316,A -85,B 0,C 180,E1 -6361.422,E2 -6361.422} C_VEL
LIN {X 0,Y 492.241,Z 320.666,A -85,B 0,C 180,E1 -6362.525,E2 -6362.525} C_VEL
LIN {X 0,Y 489.835,Z 320.97,A -85,B 0,C 180,E1 -6363.414,E2 -6363.414} C_VEL
LIN {X 0,Y 488.817,Z 321.094,A -85,B 0,C 180,E1 -6364.1,E2 -6364.1} C_VEL
LIN {X 0,Y 488.743,Z 321.101,A -85,B 0,C 180,E1 -6364.333,E2 -6364.333} C_VEL
LIN {X 0,Y 488.719,Z 321.106,A -85,B 0,C 180,E1 -6367.153,E2 -6367.153} C_VEL
LIN {X 0,Y 488.725,Z 321.107,A -85,B 0,C 180,E1 -6369.811,E2 -6369.811} C_VEL
LIN {X 0,Y 488.731,Z 321.104,A -85,B 0,C 180,E1 -6372.423,E2 -6372.423} C_VEL
LIN {X 0,Y 488.761,Z 321.104,A -85,B 0,C 180,E1 -6375,E2 -6375} C_VEL
LIN {X 0,Y 488.802,Z 321.095,A -85,B 0,C 180,E1 -6378.388,E2 -6378.388} C_VEL
LIN {X 0,Y 488.815,Z 321.096,A -85,B 0,C 180,E1 -6381.734,E2 -6381.734} C_VEL
LIN {X 0,Y 488.855,Z 321.089,A -85,B 0,C 180,E1 -6384.224,E2 -6384.224} C_VEL
LIN {X 0,Y 488.959,Z 321.078,A -85,B 0,C 180,E1 -6387.529,E2 -6387.529} C_VEL
LIN {X 0,Y 488.951,Z 321.081,A -85,B 0,C 180,E1 -6390.824,E2 -6390.824} C_VEL
LIN {X 0,Y 488.959,Z 321.078,A -85,B 0,C 180,E1 -6392.471,E2 -6392.471} C_VEL
LIN {X 0,Y 488.855,Z 321.089,A -85,B 0,C 180,E1 -6395.776,E2 -6395.776} C_VEL
LIN {X 0,Y 488.815,Z 321.096,A -85,B 0,C 180,E1 -6398.266,E2 -6398.266} C_VEL
LIN {X 0,Y 488.802,Z 321.095,A -85,B 0,C 180,E1 -6401.612,E2 -6401.612} C_VEL
LIN {X 0,Y 488.761,Z 321.104,A -85,B 0,C 180,E1 -6405,E2 -6405} C_VEL
LIN {X 0,Y 488.751,Z 321.107,A -85,B 0,C 180,E1 -6408.442,E2 -6408.442} C_VEL
LIN {X 0,Y 488.703,Z 321.107,A -85,B 0,C 180,E1 -6411.071,E2 -6411.071} C_VEL
LIN {X 0,Y 488.686,Z 321.108,A -85,B 0,C 180,E1 -6413.746,E2 -6413.746} C_VEL
LIN {X 0,Y 488.795,Z 321.095,A -85,B 0,C 180,E1 -6416.945,E2 -6416.945} C_VEL
LIN {X 0,Y 488.707,Z 321.112,A -85,B 0,C 180,E1 -6420.363,E2 -6420.363} C_VEL
LIN {X 0,Y 488.732,Z 321.102,A -85,B 0,C 180,E1 -6423.485,E2 -6423.485} C_VEL
LIN {X 0,Y 488.684,Z 321.113,A -85,B 0,C 180,E1 -6426.356,E2 -6426.356} C_VEL
LIN {X 0,Y 488.739,Z 321.101,A -85,B 0,C 180,E1 -6429.25,E2 -6429.25} C_VEL
LIN {X 0,Y 488.709,Z 321.108,A -85,B 0,C 180,E1 -6431.601,E2 -6431.601} C_VEL
LIN {X 0,Y 488.708,Z 321.105,A -85,B 0,C 180,E1 -6434.802,E2 -6434.802} C_VEL
LIN {X 0,Y 488.728,Z 321.106,A -85,B 0,C 180,E1 -6437.479,E2 -6437.479} C_VEL
LIN {X 0,Y 488.739,Z 321.101,A -85,B 0,C 180,E1 -6440.75,E2 -6440.75} C_VEL
LIN {X 0,Y 488.674,Z 321.115,A -85,B 0,C 180,E1 -6443.868,E2 -6443.868} C_VEL
LIN {X 0,Y 488.736,Z 321.102,A -85,B 0,C 180,E1 -6446.878,E2 -6446.878} C_VEL
LIN {X 0,Y 488.721,Z 321.108,A -85,B 0,C 180,E1 -6449.781,E2 -6449.781} C_VEL
LIN {X 0,Y 488.789,Z 321.098,A -85,B 0,C 180,E1 -6453.057,E2 -6453.057} C_VEL
LIN {X 0,Y 488.686,Z 321.108,A -85,B 0,C 180,E1 -6456.255,E2 -6456.255} C_VEL
LIN {X 0,Y 488.744,Z 321.107,A -85,B 0,C 180,E1 -6459.176,E2 -6459.176} C_VEL
LIN {X 0,Y 488.757,Z 321.102,A -85,B 0,C 180,E1 -6461.628,E2 -6461.628} C_VEL
LIN {X 0,Y 488.76,Z 321.104,A -85,B 0,C 180,E1 -6465,E2 -6465} C_VEL
LIN {X 0,Y 488.804,Z 321.093,A -85,B 0,C 180,E1 -6468.388,E2 -6468.388} C_VEL
LIN {X 0,Y 488.816,Z 321.092,A -85,B 0,C 180,E1 -6471.734,E2 -6471.734} C_VEL
LIN {X 0,Y 488.847,Z 321.088,A -85,B 0,C 180,E1 -6474.225,E2 -6474.225} C_VEL
LIN {X 0,Y 488.961,Z 321.074,A -85,B 0,C 180,E1 -6477.529,E2 -6477.529} C_VEL
LIN {X 0,Y 488.954,Z 321.082,A -85,B 0,C 180,E1 -6480.824,E2 -6480.824} C_VEL
LIN {X 0,Y 488.961,Z 321.078,A -85,B 0,C 180,E1 -6482.472,E2 -6482.472} C_VEL
LIN {X 0,Y 488.848,Z 321.087,A -85,B 0,C 180,E1 -6485.776,E2 -6485.776} C_VEL
LIN {X 0,Y 488.817,Z 321.095,A -85,B 0,C 180,E1 -6488.267,E2 -6488.267} C_VEL
LIN {X 0,Y 488.805,Z 321.093,A -85,B 0,C 180,E1 -6491.613,E2 -6491.613} C_VEL
LIN {X 0,Y 488.765,Z 321.099,A -85,B 0,C 180,E1 -6495.001,E2 -6495.001} C_VEL
LIN {X 0,Y 488.747,Z 321.107,A -85,B 0,C 180,E1 -6498.443,E2 -6498.443} C_VEL
LIN {X 0,Y 488.707,Z 321.105,A -85,B 0,C 180,E1 -6501.071,E2 -6501.071} C_VEL
LIN {X 0,Y 488.68,Z 321.11,A -85,B 0,C 180,E1 -6503.747,E2 -6503.747} C_VEL
LIN {X 0,Y 488.792,Z 321.095,A -85,B 0,C 180,E1 -6506.944,E2 -6506.944} C_VEL
LIN {X 0,Y 488.71,Z 321.109,A -85,B 0,C 180,E1 -6510.363,E2 -6510.363} C_VEL
LIN {X 0,Y 488.735,Z 321.103,A -85,B 0,C 180,E1 -6513.485,E2 -6513.485} C_VEL
LIN {X 0,Y 488.683,Z 321.114,A -85,B 0,C 180,E1 -6516.355,E2 -6516.355} C_VEL
LIN {X 0,Y 488.702,Z 321.111,A -85,B 0,C 180,E1 -6519.255,E2 -6519.255} C_VEL
LIN {X 0,Y 488.708,Z 321.113,A -85,B 0,C 180,E1 -6521.6,E2 -6521.6} C_VEL
LIN {X 0,Y 488.711,Z 321.305,A -85,B 0,C 180,E1 -6522.827,E2 -6522.827} C_VEL
LIN {X 0,Y 489.259,Z 325.054,A -85,B 0,C 180,E1 -6525.909,E2 -6525.909} C_VEL
LIN {X 0,Y 489.485,Z 328.197,A -85,B 0,C 180,E1 -6528.298,E2 -6528.298} C_VEL
LIN {X 0,Y 489.356,Z 331.857,A -85,B 0,C 180,E1 -6530.854,E2 -6530.854} C_VEL
LIN {X 0,Y 489.146,Z 336.518,A -85,B 0,C 180,E1 -6533.908,E2 -6533.908} C_VEL
LIN {X 0,Y 488.93,Z 341.385,A -85,B 0,C 180,E1 -6536.892,E2 -6536.892} C_VEL
LIN {X 0,Y 488.746,Z 346.323,A -85,B 0,C 180,E1 -6539.782,E2 -6539.782} C_VEL
LIN {X 0,Y 488.505,Z 352.335,A -85,B 0,C 180,E1 -6543.124,E2 -6543.124} C_VEL
LIN {X 0,Y 488.278,Z 358.187,A -85,B 0,C 180,E1 -6546.233,E2 -6546.233} C_VEL
LIN {X 0,Y 488.175,Z 364.261,A -85,B 0,C 180,E1 -6549.354,E2 -6549.354} C_VEL
LIN {X 0,Y 488.067,Z 370.366,A -85,B 0,C 180,E1 -6552.399,E2 -6552.399} C_VEL
LIN {X 0,Y 488.01,Z 376.398,A -85,B 0,C 180,E1 -6555.311,E2 -6555.311} C_VEL
LIN {X 0,Y 489.593,Z 386.473,A -85,B 0,C 180,E1 -6555.61,E2 -6555.61} C_VEL
LIN {X 0,Y 490.684,Z 394.325,A -85,B 0,C 180,E1 -6555.908,E2 -6555.908} C_VEL
LIN {X 0,Y 490.358,Z 404.972,A -85,B 0,C 180,E1 -6556.374,E2 -6556.374} C_VEL
LIN {X 0,Y 490.046,Z 415.12,A -85,B 0,C 180,E1 -6556.946,E2 -6556.946} C_VEL
LIN {X 0,Y 489.648,Z 424.115,A -85,B 0,C 180,E1 -6557.567,E2 -6557.567} C_VEL
LIN {X 0,Y 489.412,Z 432.849,A -85,B 0,C 180,E1 -6558.297,E2 -6558.297} C_VEL
LIN {X 0,Y 489.119,Z 440.247,A -85,B 0,C 180,E1 -6559.025,E2 -6559.025} C_VEL
LIN {X 0,Y 488.816,Z 447.468,A -85,B 0,C 180,E1 -6559.856,E2 -6559.856} C_VEL
LIN {X 0,Y 488.565,Z 453.671,A -85,B 0,C 180,E1 -6560.687,E2 -6560.687} C_VEL
LIN {X 0,Y 488.35,Z 460.209,A -85,B 0,C 180,E1 -6561.726,E2 -6561.726} C_VEL
LIN {X 0,Y 488.203,Z 464.71,A -85,B 0,C 180,E1 -6562.556,E2 -6562.556} C_VEL
LIN {X 0,Y 488.036,Z 470.126,A -85,B 0,C 180,E1 -6563.78,E2 -6563.78} C_VEL
LIN {X 0,Y 487.972,Z 474.521,A -85,B 0,C 180,E1 -6565.043,E2 -6565.043} C_VEL
LIN {X 0,Y 487.93,Z 476.885,A -85,B 0,C 180,E1 -6565.87,E2 -6565.87} C_VEL
LIN {X 0,Y 487.965,Z 478.682,A -85,B 0,C 180,E1 -6566.697,E2 -6566.697} C_VEL
LIN {X 0,Y 487.891,Z 481.121,A -85,B 0,C 180,E1 -6568.349,E2 -6568.349} C_VEL
LIN {X 0,Y 487.834,Z 481.707,A -85,B 0,C 180,E1 -6569.175,E2 -6569.175} C_VEL
LIN {X 0,Y 487.834,Z 481.707,A -85,B 0,C 180,E1 -6570.825,E2 -6570.825} C_VEL
LIN {X 0,Y 487.891,Z 481.121,A -85,B 0,C 180,E1 -6571.651,E2 -6571.651} C_VEL
LIN {X 0,Y 487.965,Z 478.682,A -85,B 0,C 180,E1 -6573.303,E2 -6573.303} C_VEL
LIN {X 0,Y 487.925,Z 475.736,A -85,B 0,C 180,E1 -6574.544,E2 -6574.544} C_VEL
LIN {X 0,Y 488.035,Z 471.753,A -85,B 0,C 180,E1 -6575.785,E2 -6575.785} C_VEL
LIN {X 0,Y 488.1,Z 468.54,A -85,B 0,C 180,E1 -6576.615,E2 -6576.615} C_VEL
LIN {X 0,Y 488.262,Z 462.52,A -85,B 0,C 180,E1 -6577.859,E2 -6577.859} C_VEL
LIN {X 0,Y 488.468,Z 456.423,A -85,B 0,C 180,E1 -6578.898,E2 -6578.898} C_VEL
LIN {X 0,Y 488.701,Z 450.723,A -85,B 0,C 180,E1 -6579.728,E2 -6579.728} C_VEL
LIN {X 0,Y 489.009,Z 442.166,A -85,B 0,C 180,E1 -6580.768,E2 -6580.768} C_VEL
LIN {X 0,Y 489.353,Z 433.984,A -85,B 0,C 180,E1 -6581.599,E2 -6581.599} C_VEL
LIN {X 0,Y 489.653,Z 425.469,A -85,B 0,C 180,E1 -6582.328,E2 -6582.328} C_VEL
LIN {X 0,Y 489.923,Z 417.238,A -85,B 0,C 180,E1 -6582.921,E2 -6582.921} C_VEL
LIN {X 0,Y 490.274,Z 406.986,A -85,B 0,C 180,E1 -6583.523,E2 -6583.523} C_VEL
LIN {X 0,Y 490.608,Z 398.19,A -85,B 0,C 180,E1 -6583.936,E2 -6583.936} C_VEL
LIN {X 0,Y 490.684,Z 393.036,A -85,B 0,C 180,E1 -6584.145,E2 -6584.145} C_VEL
LIN {X 0,Y 488.508,Z 379.664,A -85,B 0,C 180,E1 -6584.609,E2 -6584.609} C_VEL
LIN {X 0,Y 487.987,Z 376.341,A -85,B 0,C 180,E1 -6584.705,E2 -6584.705} C_VEL
LIN {X 0,Y 488.095,Z 369.273,A -85,B 0,C 180,E1 -6588.134,E2 -6588.134} C_VEL
LIN {X 0,Y 488.179,Z 363.366,A -85,B 0,C 180,E1 -6591.094,E2 -6591.094} C_VEL
LIN {X 0,Y 488.278,Z 358.176,A -85,B 0,C 180,E1 -6593.767,E2 -6593.767} C_VEL
LIN {X 0,Y 488.506,Z 352.327,A -85,B 0,C 180,E1 -6596.877,E2 -6596.877} C_VEL
LIN {X 0,Y 488.744,Z 346.303,A -85,B 0,C 180,E1 -6600.218,E2 -6600.218} C_VEL
LIN {X 0,Y 488.914,Z 341.353,A -85,B 0,C 180,E1 -6603.109,E2 -6603.109} C_VEL
LIN {X 0,Y 489.143,Z 336.517,A -85,B 0,C 180,E1 -6606.092,E2 -6606.092} C_VEL
LIN {X 0,Y 489.344,Z 331.773,A -85,B 0,C 180,E1 -6609.193,E2 -6609.193} C_VEL
LIN {X 0,Y 489.475,Z 328.189,A -85,B 0,C 180,E1 -6611.7,E2 -6611.7} C_VEL
LIN {X 0,Y 489.259,Z 325.019,A -85,B 0,C 180,E1 -6614.091,E2 -6614.091} C_VEL
LIN {X 0,Y 488.71,Z 321.311,A -85,B 0,C 180,E1 -6617.173,E2 -6617.173} C_VEL
LIN {X 0,Y 488.734,Z 321.108,A -85,B 0,C 180,E1 -6619.676,E2 -6619.676} C_VEL
LIN {X 0,Y 488.68,Z 321.112,A -85,B 0,C 180,E1 -6622.841,E2 -6622.841} C_VEL
LIN {X 0,Y 488.731,Z 321.111,A -85,B 0,C 180,E1 -6625.887,E2 -6625.887} C_VEL
LIN {X 0,Y 488.692,Z 321.107,A -85,B 0,C 180,E1 -6628.82,E2 -6628.82} C_VEL
LIN {X 0,Y 488.745,Z 321.106,A -85,B 0,C 180,E1 -6631.671,E2 -6631.671} C_VEL
LIN {X 0,Y 488.727,Z 321.103,A -85,B 0,C 180,E1 -6634.443,E2 -6634.443} C_VEL
LIN {X 0,Y 488.722,Z 321.104,A -85,B 0,C 180,E1 -6637.153,E2 -6637.153} C_VEL
LIN {X 0,Y 488.725,Z 321.109,A -85,B 0,C 180,E1 -6639.81,E2 -6639.81} C_VEL
LIN {X 0,Y 488.715,Z 321.104,A -85,B 0,C 180,E1 -6642.422,E2 -6642.422} C_VEL
LIN {X 0,Y 488.765,Z 321.099,A -85,B 0,C 180,E1 -6644.999,E2 -6644.999} C_VEL
LIN {X 0,Y 488.805,Z 321.093,A -85,B 0,C 180,E1 -6648.387,E2 -6648.387} C_VEL
LIN {X 0,Y 488.817,Z 321.095,A -85,B 0,C 180,E1 -6651.733,E2 -6651.733} C_VEL
LIN {X 0,Y 488.848,Z 321.087,A -85,B 0,C 180,E1 -6654.224,E2 -6654.224} C_VEL
LIN {X 0,Y 488.961,Z 321.078,A -85,B 0,C 180,E1 -6657.528,E2 -6657.528} C_VEL
LIN {X 0,Y 488.969,Z 321.072,A -85,B 0,C 180,E1 -6660,E2 -6660} C_VEL
LIN {X 0,Y 488.961,Z 321.074,A -85,B 0,C 180,E1 -6662.471,E2 -6662.471} C_VEL
LIN {X 0,Y 488.847,Z 321.088,A -85,B 0,C 180,E1 -6665.775,E2 -6665.775} C_VEL
LIN {X 0,Y 488.816,Z 321.092,A -85,B 0,C 180,E1 -6668.266,E2 -6668.266} C_VEL
LIN {X 0,Y 488.804,Z 321.093,A -85,B 0,C 180,E1 -6671.612,E2 -6671.612} C_VEL
LIN {X 0,Y 488.76,Z 321.104,A -85,B 0,C 180,E1 -6675,E2 -6675} C_VEL
LIN {X 0,Y 488.753,Z 321.103,A -85,B 0,C 180,E1 -6678.442,E2 -6678.442} C_VEL
LIN {X 0,Y 488.704,Z 321.108,A -85,B 0,C 180,E1 -6681.07,E2 -6681.07} C_VEL
LIN {X 0,Y 488.686,Z 321.108,A -85,B 0,C 180,E1 -6683.745,E2 -6683.745} C_VEL
LIN {X 0,Y 488.789,Z 321.098,A -85,B 0,C 180,E1 -6686.943,E2 -6686.943} C_VEL
LIN {X 0,Y 488.708,Z 321.112,A -85,B 0,C 180,E1 -6690.363,E2 -6690.363} C_VEL
LIN {X 0,Y 488.732,Z 321.102,A -85,B 0,C 180,E1 -6693.484,E2 -6693.484} C_VEL
LIN {X 0,Y 488.684,Z 321.115,A -85,B 0,C 180,E1 -6696.355,E2 -6696.355} C_VEL
LIN {X 0,Y 488.739,Z 321.101,A -85,B 0,C 180,E1 -6699.25,E2 -6699.25} C_VEL
LIN {X 0,Y 488.728,Z 321.106,A -85,B 0,C 180,E1 -6702.521,E2 -6702.521} C_VEL
LIN {X 0,Y 488.708,Z 321.105,A -85,B 0,C 180,E1 -6705.198,E2 -6705.198} C_VEL
LIN {X 0,Y 488.709,Z 321.108,A -85,B 0,C 180,E1 -6708.399,E2 -6708.399} C_VEL
LIN {X 0,Y 488.737,Z 321.101,A -85,B 0,C 180,E1 -6710.942,E2 -6710.942} C_VEL
LIN {X 0,Y 488.68,Z 321.117,A -85,B 0,C 180,E1 -6713.868,E2 -6713.868} C_VEL
LIN {X 0,Y 488.735,Z 321.101,A -85,B 0,C 180,E1 -6716.877,E2 -6716.877} C_VEL
LIN {X 0,Y 488.72,Z 321.111,A -85,B 0,C 180,E1 -6719.781,E2 -6719.781} C_VEL
LIN {X 0,Y 488.795,Z 321.095,A -85,B 0,C 180,E1 -6723.055,E2 -6723.055} C_VEL
LIN {X 0,Y 488.743,Z 321.101,A -85,B 0,C 180,E1 -6724.333,E2 -6724.333} C_VEL
LIN {X 0,Y 488.094,Z 321.184,A -85,B 0,C 180,E1 -6725.02,E2 -6725.02} C_VEL
LIN {X 0,Y 485.225,Z 321.545,A -85,B 0,C 180,E1 -6726.137,E2 -6726.137} C_VEL
LIN {X 0,Y 482.78,Z 321.851,A -85,B 0,C 180,E1 -6727.036,E2 -6727.036} C_VEL
LIN {X 0,Y 481.722,Z 321.981,A -85,B 0,C 180,E1 -6727.732,E2 -6727.732} C_VEL
LIN {X 0,Y 481.632,Z 321.989,A -85,B 0,C 180,E1 -6727.967,E2 -6727.967} C_VEL
LIN {X 0,Y 481.704,Z 321.977,A -85,B 0,C 180,E1 -6730.393,E2 -6730.393} C_VEL
LIN {X 0,Y 481.688,Z 321.985,A -85,B 0,C 180,E1 -6733.034,E2 -6733.034} C_VEL
LIN {X 0,Y 481.691,Z 321.985,A -85,B 0,C 180,E1 -6735.639,E2 -6735.639} C_VEL
LIN {X 0,Y 481.748,Z 321.974,A -85,B 0,C 180,E1 -6738.215,E2 -6738.215} C_VEL
LIN {X 0,Y 481.76,Z 321.976,A -85,B 0,C 180,E1 -6741.612,E2 -6741.612} C_VEL
LIN {X 0,Y 481.816,Z 321.966,A -85,B 0,C 180,E1 -6744.14,E2 -6744.14} C_VEL
LIN {X 0,Y 481.926,Z 321.955,A -85,B 0,C 180,E1 -6747.493,E2 -6747.493} C_VEL
LIN {X 0,Y 481.902,Z 321.959,A -85,B 0,C 180,E1 -6750.836,E2 -6750.836} C_VEL
LIN {X 0,Y 481.926,Z 321.955,A -85,B 0,C 180,E1 -6752.507,E2 -6752.507} C_VEL
LIN {X 0,Y 481.816,Z 321.966,A -85,B 0,C 180,E1 -6755.86,E2 -6755.86} C_VEL
LIN {X 0,Y 481.76,Z 321.976,A -85,B 0,C 180,E1 -6758.388,E2 -6758.388} C_VEL
LIN {X 0,Y 481.748,Z 321.974,A -85,B 0,C 180,E1 -6761.785,E2 -6761.785} C_VEL
LIN {X 0,Y 481.741,Z 321.977,A -85,B 0,C 180,E1 -6765.224,E2 -6765.224} C_VEL
LIN {X 0,Y 481.709,Z 321.984,A -85,B 0,C 180,E1 -6768.722,E2 -6768.722} C_VEL
LIN {X 0,Y 481.642,Z 321.985,A -85,B 0,C 180,E1 -6771.395,E2 -6771.395} C_VEL
LIN {X 0,Y 481.671,Z 321.986,A -85,B 0,C 180,E1 -6774.113,E2 -6774.113} C_VEL
LIN {X 0,Y 481.749,Z 321.972,A -85,B 0,C 180,E1 -6777.141,E2 -6777.141} C_VEL
LIN {X 0,Y 481.675,Z 321.983,A -85,B 0,C 180,E1 -6779.741,E2 -6779.741} C_VEL
LIN {X 0,Y 481.67,Z 321.984,A -85,B 0,C 180,E1 -6782.674,E2 -6782.674} C_VEL
LIN {X 0,Y 481.638,Z 321.988,A -85,B 0,C 180,E1 -6785.709,E2 -6785.709} C_VEL
LIN {X 0,Y 481.711,Z 321.977,A -85,B 0,C 180,E1 -6789.354,E2 -6789.354} C_VEL
LIN {X 0,Y 481.645,Z 321.99,A -85,B 0,C 180,E1 -6792.161,E2 -6792.161} C_VEL
LIN {X 0,Y 481.657,Z 321.987,A -85,B 0,C 180,E1 -6795.543,E2 -6795.543} C_VEL
LIN {X 0,Y 481.67,Z 321.986,A -85,B 0,C 180,E1 -6798.085,E2 -6798.085} C_VEL
LIN {X 0,Y 481.694,Z 321.98,A -85,B 0,C 180,E1 -6801.144,E2 -6801.144} C_VEL
LIN {X 0,Y 481.659,Z 321.983,A -85,B 0,C 180,E1 -6804.796,E2 -6804.796} C_VEL
LIN {X 0,Y 481.67,Z 321.986,A -85,B 0,C 180,E1 -6807.326,E2 -6807.326} C_VEL
LIN {X 0,Y 481.676,Z 321.981,A -85,B 0,C 180,E1 -6810.259,E2 -6810.259} C_VEL
LIN {X 0,Y 481.743,Z 321.976,A -85,B 0,C 180,E1 -6813.112,E2 -6813.112} C_VEL
LIN {X 0,Y 481.671,Z 321.984,A -85,B 0,C 180,E1 -6815.887,E2 -6815.887} C_VEL
LIN {X 0,Y 481.7,Z 321.982,A -85,B 0,C 180,E1 -6819.028,E2 -6819.028} C_VEL
LIN {X 0,Y 481.705,Z 321.977,A -85,B 0,C 180,E1 -6822.159,E2 -6822.159} C_VEL
LIN {X 0,Y 481.741,Z 321.976,A -85,B 0,C 180,E1 -6824.776,E2 -6824.776} C_VEL
LIN {X 0,Y 481.749,Z 321.972,A -85,B 0,C 180,E1 -6828.216,E2 -6828.216} C_VEL
LIN {X 0,Y 481.761,Z 321.971,A -85,B 0,C 180,E1 -6831.612,E2 -6831.612} C_VEL
LIN {X 0,Y 481.807,Z 321.965,A -85,B 0,C 180,E1 -6834.14,E2 -6834.14} C_VEL
LIN {X 0,Y 481.927,Z 321.951,A -85,B 0,C 180,E1 -6837.493,E2 -6837.493} C_VEL
LIN {X 0,Y 481.905,Z 321.96,A -85,B 0,C 180,E1 -6840.836,E2 -6840.836} C_VEL
LIN {X 0,Y 481.927,Z 321.954,A -85,B 0,C 180,E1 -6842.508,E2 -6842.508} C_VEL
LIN {X 0,Y 481.808,Z 321.964,A -85,B 0,C 180,E1 -6845.861,E2 -6845.861} C_VEL
LIN {X 0,Y 481.763,Z 321.975,A -85,B 0,C 180,E1 -6848.389,E2 -6848.389} C_VEL
LIN {X 0,Y 481.751,Z 321.972,A -85,B 0,C 180,E1 -6851.785,E2 -6851.785} C_VEL
LIN {X 0,Y 481.744,Z 321.973,A -85,B 0,C 180,E1 -6855.225,E2 -6855.225} C_VEL
LIN {X 0,Y 481.708,Z 321.98,A -85,B 0,C 180,E1 -6858.722,E2 -6858.722} C_VEL
LIN {X 0,Y 481.645,Z 321.984,A -85,B 0,C 180,E1 -6861.395,E2 -6861.395} C_VEL
LIN {X 0,Y 481.661,Z 321.989,A -85,B 0,C 180,E1 -6864.114,E2 -6864.114} C_VEL
LIN {X 0,Y 481.747,Z 321.972,A -85,B 0,C 180,E1 -6867.14,E2 -6867.14} C_VEL
LIN {X 0,Y 481.679,Z 321.984,A -85,B 0,C 180,E1 -6869.742,E2 -6869.742} C_VEL
LIN {X 0,Y 481.672,Z 321.982,A -85,B 0,C 180,E1 -6872.675,E2 -6872.675} C_VEL
LIN {X 0,Y 481.637,Z 321.99,A -85,B 0,C 180,E1 -6875.71,E2 -6875.71} C_VEL
LIN {X 0,Y 481.672,Z 321.986,A -85,B 0,C 180,E1 -6878.859,E2 -6878.859} C_VEL
LIN {X 0,Y 481.653,Z 321.992,A -85,B 0,C 180,E1 -6881.913,E2 -6881.913} C_VEL
LIN {X 0,Y 481.795,Z 323.039,A -85,B 0,C 180,E1 -6883.283,E2 -6883.283} C_VEL
LIN {X 0,Y 482.199,Z 325.82,A -85,B 0,C 180,E1 -6885.606,E2 -6885.606} C_VEL
LIN {X 0,Y 482.477,Z 328.875,A -85,B 0,C 180,E1 -6887.979,E2 -6887.979} C_VEL
LIN {X 0,Y 482.336,Z 332.502,A -85,B 0,C 180,E1 -6890.557,E2 -6890.557} C_VEL
LIN {X 0,Y 482.179,Z 336.573,A -85,B 0,C 180,E1 -6893.302,E2 -6893.302} C_VEL
LIN {X 0,Y 481.941,Z 341.404,A -85,B 0,C 180,E1 -6896.349,E2 -6896.349} C_VEL
LIN {X 0,Y 481.687,Z 346.527,A -85,B 0,C 180,E1 -6899.411,E2 -6899.411} C_VEL
LIN {X 0,Y 481.482,Z 351.32,A -85,B 0,C 180,E1 -6902.155,E2 -6902.155} C_VEL
LIN {X 0,Y 481.325,Z 356.409,A -85,B 0,C 180,E1 -6904.948,E2 -6904.948} C_VEL
LIN {X 0,Y 481.161,Z 361.561,A -85,B 0,C 180,E1 -6907.681,E2 -6907.681} C_VEL
LIN {X 0,Y 481.033,Z 366.751,A -85,B 0,C 180,E1 -6910.365,E2 -6910.365} C_VEL
LIN {X 0,Y 480.926,Z 371.979,A -85,B 0,C 180,E1 -6913.006,E2 -6913.006} C_VEL
LIN {X 0,Y 480.942,Z 376.28,A -85,B 0,C 180,E1 -6915.092,E2 -6915.092} C_VEL
LIN {X 0,Y 482.638,Z 386.713,A -85,B 0,C 180,E1 -6915.412,E2 -6915.412} C_VEL
LIN {X 0,Y 483.775,Z 395.418,A -85,B 0,C 180,E1 -6915.756,E2 -6915.756} C_VEL
LIN {X 0,Y 483.464,Z 404.776,A -85,B 0,C 180,E1 -6916.176,E2 -6916.176} C_VEL
LIN {X 0,Y 483.117,Z 414.924,A -85,B 0,C 180,E1 -6916.755,E2 -6916.755} C_VEL
LIN {X 0,Y 482.688,Z 423.918,A -85,B 0,C 180,E1 -6917.385,E2 -6917.385} C_VEL
LIN {X 0,Y 482.44,Z 432.682,A -85,B 0,C 180,E1 -6918.128,E2 -6918.128} C_VEL
LIN {X 0,Y 482.136,Z 440.051,A -85,B 0,C 180,E1 -6918.864,E2 -6918.864} C_VEL
LIN {X 0,Y 481.782,Z 447.271,A -85,B 0,C 180,E1 -6919.706,E2 -6919.706} C_VEL
LIN {X 0,Y 481.513,Z 453.474,A -85,B 0,C 180,E1 -6920.549,E2 -6920.549} C_VEL
LIN {X 0,Y 481.308,Z 460.013,A -85,B 0,C 180,E1 -6921.604,E2 -6921.604} C_VEL
LIN {X 0,Y 481.137,Z 464.514,A -85,B 0,C 180,E1 -6922.446,E2 -6922.446} C_VEL
LIN {X 0,Y 480.936,Z 470.388,A -85,B 0,C 180,E1 -6923.812,E2 -6923.812} C_VEL
LIN {X 0,Y 480.902,Z 474.325,A -85,B 0,C 180,E1 -6924.97,E2 -6924.97} C_VEL
LIN {X 0,Y 480.83,Z 476.689,A -85,B 0,C 180,E1 -6925.809,E2 -6925.809} C_VEL
LIN {X 0,Y 480.889,Z 478.487,A -85,B 0,C 180,E1 -6926.649,E2 -6926.649} C_VEL
LIN {X 0,Y 480.793,Z 480.925,A -85,B 0,C 180,E1 -6928.325,E2 -6928.325} C_VEL
LIN {X 0,Y 480.76,Z 481.512,A -85,B 0,C 180,E1 -6929.162,E2 -6929.162} C_VEL
LIN {X 0,Y 480.76,Z 481.512,A -85,B 0,C 180,E1 -6930.838,E2 -6930.838} C_VEL
LIN {X 0,Y 480.793,Z 480.925,A -85,B 0,C 180,E1 -6931.675,E2 -6931.675} C_VEL
LIN {X 0,Y 480.889,Z 478.487,A -85,B 0,C 180,E1 -6933.351,E2 -6933.351} C_VEL
LIN {X 0,Y 480.843,Z 475.54,A -85,B 0,C 180,E1 -6934.611,E2 -6934.611} C_VEL
LIN {X 0,Y 480.939,Z 471.556,A -85,B 0,C 180,E1 -6935.871,E2 -6935.871} C_VEL
LIN {X 0,Y 481.016,Z 468.344,A -85,B 0,C 180,E1 -6936.712,E2 -6936.712} C_VEL
LIN {X 0,Y 481.21,Z 462.323,A -85,B 0,C 180,E1 -6937.975,E2 -6937.975} C_VEL
LIN {X 0,Y 481.418,Z 456.226,A -85,B 0,C 180,E1 -6939.029,E2 -6939.029} C_VEL
LIN {X 0,Y 481.675,Z 450.526,A -85,B 0,C 180,E1 -6939.872,E2 -6939.872} C_VEL
LIN {X 0,Y 482.028,Z 441.97,A -85,B 0,C 180,E1 -6940.926,E2 -6940.926} C_VEL
LIN {X 0,Y 482.381,Z 433.788,A -85,B 0,C 180,E1 -6941.769,E2 -6941.769} C_VEL
LIN {X 0,Y 482.659,Z 425.232,A -85,B 0,C 180,E1 -6942.512,E2 -6942.512} C_VEL
LIN {X 0,Y 482.972,Z 417.041,A -85,B 0,C 180,E1 -6943.11,E2 -6943.11} C_VEL
LIN {X 0,Y 483.361,Z 406.79,A -85,B 0,C 180,E1 -6943.72,E2 -6943.72} C_VEL
LIN {X 0,Y 483.719,Z 397.995,A -85,B 0,C 180,E1 -6944.139,E2 -6944.139} C_VEL
LIN {X 0,Y 483.563,Z 392.834,A -85,B 0,C 180,E1 -6944.358,E2 -6944.358} C_VEL
LIN {X 0,Y 481.304,Z 378.792,A -85,B 0,C 180,E1 -6944.846,E2 -6944.846} C_VEL
LIN {X 0,Y 480.921,Z 376.181,A -85,B 0,C 180,E1 -6944.926,E2 -6944.926} C_VEL
LIN {X 0,Y 481.012,Z 369.475,A -85,B 0,C 180,E1 -6948.248,E2 -6948.248} C_VEL
LIN {X 0,Y 481.108,Z 363.265,A -85,B 0,C 180,E1 -6951.42,E2 -6951.42} C_VEL
LIN {X 0,Y 481.238,Z 358.106,A -85,B 0,C 180,E1 -6954.136,E2 -6954.136} C_VEL
LIN {X 0,Y 481.446,Z 352.712,A -85,B 0,C 180,E1 -6957.068,E2 -6957.068} C_VEL
LIN {X 0,Y 481.62,Z 347.956,A -85,B 0,C 180,E1 -6959.745,E2 -6959.745} C_VEL
LIN {X 0,Y 481.845,Z 342.993,A -85,B 0,C 180,E1 -6962.661,E2 -6962.661} C_VEL
LIN {X 0,Y 482.062,Z 338.157,A -85,B 0,C 180,E1 -6965.673,E2 -6965.673} C_VEL
LIN {X 0,Y 482.277,Z 333.393,A -85,B 0,C 180,E1 -6968.801,E2 -6968.801} C_VEL
LIN {X 0,Y 482.431,Z 330.318,A -85,B 0,C 180,E1 -6970.962,E2 -6970.962} C_VEL
LIN {X 0,Y 482.399,Z 327.248,A -85,B 0,C 180,E1 -6973.243,E2 -6973.243} C_VEL
LIN {X 0,Y 481.961,Z 324.335,A -85,B 0,C 180,E1 -6975.604,E2 -6975.604} C_VEL
LIN {X 0,Y 481.649,Z 321.991,A -85,B 0,C 180,E1 -6977.839,E2 -6977.839} C_VEL
LIN {X 0,Y 481.681,Z 321.986,A -85,B 0,C 180,E1 -6980.651,E2 -6980.651} C_VEL
LIN {X 0,Y 481.628,Z 321.991,A -85,B 0,C 180,E1 -6983.376,E2 -6983.376} C_VEL
LIN {X 0,Y 481.711,Z 321.98,A -85,B 0,C 180,E1 -6986.33,E2 -6986.33} C_VEL
LIN {X 0,Y 481.651,Z 321.986,A -85,B 0,C 180,E1 -6989.417,E2 -6989.417} C_VEL
LIN {X 0,Y 481.7,Z 321.982,A -85,B 0,C 180,E1 -6992.168,E2 -6992.168} C_VEL
LIN {X 0,Y 481.693,Z 321.979,A -85,B 0,C 180,E1 -6994.968,E2 -6994.968} C_VEL
LIN {X 0,Y 481.649,Z 321.992,A -85,B 0,C 180,E1 -6997.704,E2 -6997.704} C_VEL
LIN {X 0,Y 481.704,Z 321.978,A -85,B 0,C 180,E1 -7000.393,E2 -7000.393} C_VEL
LIN {X 0,Y 481.679,Z 321.982,A -85,B 0,C 180,E1 -7003.033,E2 -7003.033} C_VEL
LIN {X 0,Y 481.694,Z 321.985,A -85,B 0,C 180,E1 -7005.638,E2 -7005.638} C_VEL
LIN {X 0,Y 481.751,Z 321.972,A -85,B 0,C 180,E1 -7008.215,E2 -7008.215} C_VEL
LIN {X 0,Y 481.763,Z 321.975,A -85,B 0,C 180,E1 -7011.611,E2 -7011.611} C_VEL
LIN {X 0,Y 481.808,Z 321.964,A -85,B 0,C 180,E1 -7014.139,E2 -7014.139} C_VEL
LIN {X 0,Y 481.927,Z 321.954,A -85,B 0,C 180,E1 -7017.492,E2 -7017.492} C_VEL
LIN {X 0,Y 481.94,Z 321.948,A -85,B 0,C 180,E1 -7020,E2 -7020} C_VEL
LIN {X 0,Y 481.927,Z 321.951,A -85,B 0,C 180,E1 -7022.507,E2 -7022.507} C_VEL
LIN {X 0,Y 481.807,Z 321.965,A -85,B 0,C 180,E1 -7025.86,E2 -7025.86} C_VEL
LIN {X 0,Y 481.761,Z 321.971,A -85,B 0,C 180,E1 -7028.388,E2 -7028.388} C_VEL
LIN {X 0,Y 481.749,Z 321.972,A -85,B 0,C 180,E1 -7031.784,E2 -7031.784} C_VEL
LIN {X 0,Y 481.741,Z 321.976,A -85,B 0,C 180,E1 -7035.224,E2 -7035.224} C_VEL
LIN {X 0,Y 481.71,Z 321.985,A -85,B 0,C 180,E1 -7038.721,E2 -7038.721} C_VEL
LIN {X 0,Y 481.643,Z 321.985,A -85,B 0,C 180,E1 -7041.394,E2 -7041.394} C_VEL
LIN {X 0,Y 481.671,Z 321.984,A -85,B 0,C 180,E1 -7044.113,E2 -7044.113} C_VEL
LIN {X 0,Y 481.744,Z 321.973,A -85,B 0,C 180,E1 -7047.139,E2 -7047.139} C_VEL
LIN {X 0,Y 481.676,Z 321.981,A -85,B 0,C 180,E1 -7049.741,E2 -7049.741} C_VEL
LIN {X 0,Y 481.67,Z 321.986,A -85,B 0,C 180,E1 -7052.674,E2 -7052.674} C_VEL
LIN {X 0,Y 481.638,Z 321.987,A -85,B 0,C 180,E1 -7055.709,E2 -7055.709} C_VEL
LIN {X 0,Y 481.711,Z 321.976,A -85,B 0,C 180,E1 -7059.354,E2 -7059.354} C_VEL
LIN {X 0,Y 481.67,Z 321.99,A -85,B 0,C 180,E1 -7062.158,E2 -7062.158} C_VEL
LIN {X 0,Y 481.657,Z 321.987,A -85,B 0,C 180,E1 -7064.457,E2 -7064.457} C_VEL
LIN {X 0,Y 481.645,Z 321.99,A -85,B 0,C 180,E1 -7067.839,E2 -7067.839} C_VEL
LIN {X 0,Y 481.711,Z 321.977,A -85,B 0,C 180,E1 -7070.646,E2 -7070.646} C_VEL
LIN {X 0,Y 481.638,Z 321.988,A -85,B 0,C 180,E1 -7074.291,E2 -7074.291} C_VEL
LIN {X 0,Y 481.67,Z 321.984,A -85,B 0,C 180,E1 -7077.326,E2 -7077.326} C_VEL
LIN {X 0,Y 481.675,Z 321.983,A -85,B 0,C 180,E1 -7080.259,E2 -7080.259} C_VEL
LIN {X 0,Y 481.749,Z 321.973,A -85,B 0,C 180,E1 -7083.112,E2 -7083.112} C_VEL
LIN {X 0,Y 481.671,Z 321.986,A -85,B 0,C 180,E1 -7085.887,E2 -7085.887} C_VEL
LIN {X 0,Y 481.632,Z 321.989,A -85,B 0,C 180,E1 -7087.967,E2 -7087.967} C_VEL
LIN {X 0,Y 480.964,Z 322.07,A -85,B 0,C 180,E1 -7088.665,E2 -7088.665} C_VEL
LIN {X 0,Y 478.138,Z 322.426,A -85,B 0,C 180,E1 -7089.8,E2 -7089.8} C_VEL
LIN {X 0,Y 475.755,Z 322.726,A -85,B 0,C 180,E1 -7090.714,E2 -7090.714} C_VEL
LIN {X 0,Y 474.734,Z 322.854,A -85,B 0,C 180,E1 -7091.42,E2 -7091.42} C_VEL
LIN {X 0,Y 474.652,Z 322.862,A -85,B 0,C 180,E1 -7091.659,E2 -7091.659} C_VEL
LIN {X 0,Y 474.697,Z 322.853,A -85,B 0,C 180,E1 -7094.544,E2 -7094.544} C_VEL
LIN {X 0,Y 474.701,Z 322.852,A -85,B 0,C 180,E1 -7098.038,E2 -7098.038} C_VEL
LIN {X 0,Y 474.725,Z 322.853,A -85,B 0,C 180,E1 -7101.486,E2 -7101.486} C_VEL
LIN {X 0,Y 474.778,Z 322.843,A -85,B 0,C 180,E1 -7104.052,E2 -7104.052} C_VEL
LIN {X 0,Y 474.892,Z 322.832,A -85,B 0,C 180,E1 -7107.455,E2 -7107.455} C_VEL
LIN {X 0,Y 474.909,Z 322.828,A -85,B 0,C 180,E1 -7110,E2 -7110} C_VEL
LIN {X 0,Y 474.892,Z 322.832,A -85,B 0,C 180,E1 -7112.545,E2 -7112.545} C_VEL
LIN {X 0,Y 474.778,Z 322.843,A -85,B 0,C 180,E1 -7115.948,E2 -7115.948} C_VEL
LIN {X 0,Y 474.725,Z 322.853,A -85,B 0,C 180,E1 -7118.514,E2 -7118.514} C_VEL
LIN {X 0,Y 474.701,Z 322.852,A -85,B 0,C 180,E1 -7121.962,E2 -7121.962} C_VEL
LIN {X 0,Y 474.697,Z 322.853,A -85,B 0,C 180,E1 -7125.456,E2 -7125.456} C_VEL
LIN {X 0,Y 474.662,Z 322.858,A -85,B 0,C 180,E1 -7129.01,E2 -7129.01} C_VEL
LIN {X 0,Y 474.585,Z 322.865,A -85,B 0,C 180,E1 -7131.729,E2 -7131.729} C_VEL
LIN {X 0,Y 474.654,Z 322.863,A -85,B 0,C 180,E1 -7134.493,E2 -7134.493} C_VEL
LIN {X 0,Y 474.695,Z 322.85,A -85,B 0,C 180,E1 -7137.339,E2 -7137.339} C_VEL
LIN {X 0,Y 474.601,Z 322.864,A -85,B 0,C 180,E1 -7140.811,E2 -7140.811} C_VEL
LIN {X 0,Y 474.635,Z 322.863,A -85,B 0,C 180,E1 -7143.984,E2 -7143.984} C_VEL
LIN {X 0,Y 474.571,Z 322.866,A -85,B 0,C 180,E1 -7146.9,E2 -7146.9} C_VEL
LIN {X 0,Y 474.647,Z 322.859,A -85,B 0,C 180,E1 -7149.651,E2 -7149.651} C_VEL
LIN {X 0,Y 474.611,Z 322.861,A -85,B 0,C 180,E1 -7152.934,E2 -7152.934} C_VEL
LIN {X 0,Y 474.615,Z 322.869,A -85,B 0,C 180,E1 -7155.896,E2 -7155.896} C_VEL
LIN {X 0,Y 474.642,Z 322.857,A -85,B 0,C 180,E1 -7159.038,E2 -7159.038} C_VEL
LIN {X 0,Y 474.613,Z 322.868,A -85,B 0,C 180,E1 -7161.703,E2 -7161.703} C_VEL
LIN {X 0,Y 474.621,Z 322.86,A -85,B 0,C 180,E1 -7164.726,E2 -7164.726} C_VEL
LIN {X 0,Y 474.635,Z 322.863,A -85,B 0,C 180,E1 -7167.788,E2 -7167.788} C_VEL
LIN {X 0,Y 474.621,Z 322.861,A -85,B 0,C 180,E1 -7170.885,E2 -7170.885} C_VEL
LIN {X 0,Y 474.658,Z 322.861,A -85,B 0,C 180,E1 -7173.629,E2 -7173.629} C_VEL
LIN {X 0,Y 474.633,Z 322.859,A -85,B 0,C 180,E1 -7176.642,E2 -7176.642} C_VEL
LIN {X 0,Y 474.654,Z 322.856,A -85,B 0,C 180,E1 -7180.09,E2 -7180.09} C_VEL
LIN {X 0,Y 474.648,Z 322.859,A -85,B 0,C 180,E1 -7182.775,E2 -7182.775} C_VEL
LIN {X 0,Y 474.646,Z 322.861,A -85,B 0,C 180,E1 -7185.421,E2 -7185.421} C_VEL
LIN {X 0,Y 474.702,Z 322.849,A -85,B 0,C 180,E1 -7188.038,E2 -7188.038} C_VEL
LIN {X 0,Y 474.726,Z 322.849,A -85,B 0,C 180,E1 -7191.487,E2 -7191.487} C_VEL
LIN {X 0,Y 474.77,Z 322.841,A -85,B 0,C 180,E1 -7194.053,E2 -7194.053} C_VEL
LIN {X 0,Y 474.893,Z 322.827,A -85,B 0,C 180,E1 -7197.456,E2 -7197.456} C_VEL
LIN {X 0,Y 474.911,Z 322.824,A -85,B 0,C 180,E1 -7200,E2 -7200} C_VEL
LIN {X 0,Y 474.893,Z 322.831,A -85,B 0,C 180,E1 -7202.545,E2 -7202.545} C_VEL
LIN {X 0,Y 474.771,Z 322.841,A -85,B 0,C 180,E1 -7205.948,E2 -7205.948} C_VEL
LIN {X 0,Y 474.728,Z 322.853,A -85,B 0,C 180,E1 -7208.514,E2 -7208.514} C_VEL
LIN {X 0,Y 474.704,Z 322.851,A -85,B 0,C 180,E1 -7211.963,E2 -7211.963} C_VEL
LIN {X 0,Y 474.7,Z 322.85,A -85,B 0,C 180,E1 -7215.456,E2 -7215.456} C_VEL
LIN {X 0,Y 474.663,Z 322.855,A -85,B 0,C 180,E1 -7219.011,E2 -7219.011} C_VEL
LIN {X 0,Y 474.588,Z 322.865,A -85,B 0,C 180,E1 -7221.729,E2 -7221.729} C_VEL
LIN {X 0,Y 474.641,Z 322.862,A -85,B 0,C 180,E1 -7224.494,E2 -7224.494} C_VEL
LIN {X 0,Y 474.682,Z 322.852,A -85,B 0,C 180,E1 -7227.335,E2 -7227.335} C_VEL
LIN {X 0,Y 474.606,Z 322.868,A -85,B 0,C 180,E1 -7230.231,E2 -7230.231} C_VEL
LIN {X 0,Y 474.643,Z 322.857,A -85,B 0,C 180,E1 -7233.22,E2 -7233.22} C_VEL
LIN {X 0,Y 474.59,Z 322.87,A -85,B 0,C 180,E1 -7236.324,E2 -7236.324} C_VEL
LIN {X 0,Y 474.629,Z 322.866,A -85,B 0,C 180,E1 -7239.648,E2 -7239.648} C_VEL
LIN {X 0,Y 474.63,Z 323.053,A -85,B 0,C 180,E1 -7242.238,E2 -7242.238} C_VEL
LIN {X 0,Y 475.111,Z 326.522,A -85,B 0,C 180,E1 -7245.238,E2 -7245.238} C_VEL
LIN {X 0,Y 475.432,Z 329.578,A -85,B 0,C 180,E1 -7247.657,E2 -7247.657} C_VEL
LIN {X 0,Y 475.318,Z 333.113,A -85,B 0,C 180,E1 -7250.253,E2 -7250.253} C_VEL
LIN {X 0,Y 475.173,Z 337.132,A -85,B 0,C 180,E1 -7253.005,E2 -7253.005} C_VEL
LIN {X 0,Y 474.931,Z 341.693,A -85,B 0,C 180,E1 -7255.964,E2 -7255.964} C_VEL
LIN {X 0,Y 474.668,Z 346.323,A -85,B 0,C 180,E1 -7258.788,E2 -7258.788} C_VEL
LIN {X 0,Y 474.463,Z 351.291,A -85,B 0,C 180,E1 -7261.706,E2 -7261.706} C_VEL
LIN {X 0,Y 474.257,Z 356.582,A -85,B 0,C 180,E1 -7264.684,E2 -7264.684} C_VEL
LIN {X 0,Y 474.101,Z 361.463,A -85,B 0,C 180,E1 -7267.33,E2 -7267.33} C_VEL
LIN {X 0,Y 473.957,Z 366.641,A -85,B 0,C 180,E1 -7270.059,E2 -7270.059} C_VEL
LIN {X 0,Y 473.854,Z 371.844,A -85,B 0,C 180,E1 -7272.745,E2 -7272.745} C_VEL
LIN {X 0,Y 473.826,Z 376.054,A -85,B 0,C 180,E1 -7274.862,E2 -7274.862} C_VEL
LIN {X 0,Y 475.604,Z 386.733,A -85,B 0,C 180,E1 -7275.198,E2 -7275.198} C_VEL
LIN {X 0,Y 476.875,Z 395.221,A -85,B 0,C 180,E1 -7275.545,E2 -7275.545} C_VEL
LIN {X 0,Y 476.547,Z 404.579,A -85,B 0,C 180,E1 -7275.971,E2 -7275.971} C_VEL
LIN {X 0,Y 476.17,Z 415.051,A -85,B 0,C 180,E1 -7276.58,E2 -7276.58} C_VEL
LIN {X 0,Y 475.718,Z 423.721,A -85,B 0,C 180,E1 -7277.197,E2 -7277.197} C_VEL
LIN {X 0,Y 475.47,Z 432.592,A -85,B 0,C 180,E1 -7277.962,E2 -7277.962} C_VEL
LIN {X 0,Y 475.138,Z 439.854,A -85,B 0,C 180,E1 -7278.698,E2 -7278.698} C_VEL
LIN {X 0,Y 474.768,Z 447.074,A -85,B 0,C 180,E1 -7279.552,E2 -7279.552} C_VEL
LIN {X 0,Y 474.485,Z 453.277,A -85,B 0,C 180,E1 -7280.408,E2 -7280.408} C_VEL
LIN {X 0,Y 474.269,Z 459.816,A -85,B 0,C 180,E1 -7281.478,E2 -7281.478} C_VEL
LIN {X 0,Y 474.065,Z 464.317,A -85,B 0,C 180,E1 -7282.332,E2 -7282.332} C_VEL
LIN {X 0,Y 473.895,Z 469.507,A -85,B 0,C 180,E1 -7283.532,E2 -7283.532} C_VEL
LIN {X 0,Y 473.833,Z 474.13,A -85,B 0,C 180,E1 -7284.894,E2 -7284.894} C_VEL
LIN {X 0,Y 473.737,Z 476.492,A -85,B 0,C 180,E1 -7285.746,E2 -7285.746} C_VEL
LIN {X 0,Y 473.796,Z 478.291,A -85,B 0,C 180,E1 -7286.598,E2 -7286.598} C_VEL
LIN {X 0,Y 473.698,Z 480.73,A -85,B 0,C 180,E1 -7288.3,E2 -7288.3} C_VEL
LIN {X 0,Y 473.688,Z 481.317,A -85,B 0,C 180,E1 -7289.15,E2 -7289.15} C_VEL
LIN {X 0,Y 473.688,Z 481.317,A -85,B 0,C 180,E1 -7290.85,E2 -7290.85} C_VEL
LIN {X 0,Y 473.698,Z 480.73,A -85,B 0,C 180,E1 -7291.7,E2 -7291.7} C_VEL
LIN {X 0,Y 473.796,Z 478.291,A -85,B 0,C 180,E1 -7293.402,E2 -7293.402} C_VEL
LIN {X 0,Y 473.766,Z 475.344,A -85,B 0,C 180,E1 -7294.68,E2 -7294.68} C_VEL
LIN {X 0,Y 473.846,Z 471.359,A -85,B 0,C 180,E1 -7295.959,E2 -7295.959} C_VEL
LIN {X 0,Y 474.012,Z 466.233,A -85,B 0,C 180,E1 -7297.24,E2 -7297.24} C_VEL
LIN {X 0,Y 474.195,Z 460.971,A -85,B 0,C 180,E1 -7298.309,E2 -7298.309} C_VEL
LIN {X 0,Y 474.414,Z 454.653,A -85,B 0,C 180,E1 -7299.378,E2 -7299.378} C_VEL
LIN {X 0,Y 474.67,Z 448.701,A -85,B 0,C 180,E1 -7300.234,E2 -7300.234} C_VEL
LIN {X 0,Y 475.046,Z 441.774,A -85,B 0,C 180,E1 -7301.089,E2 -7301.089} C_VEL
LIN {X 0,Y 475.413,Z 433.591,A -85,B 0,C 180,E1 -7301.944,E2 -7301.944} C_VEL
LIN {X 0,Y 475.683,Z 425.035,A -85,B 0,C 180,E1 -7302.699,E2 -7302.699} C_VEL
LIN {X 0,Y 476.047,Z 416.845,A -85,B 0,C 180,E1 -7303.304,E2 -7303.304} C_VEL
LIN {X 0,Y 476.456,Z 406.593,A -85,B 0,C 180,E1 -7303.923,E2 -7303.923} C_VEL
LIN {X 0,Y 476.826,Z 397.798,A -85,B 0,C 180,E1 -7304.347,E2 -7304.347} C_VEL
LIN {X 0,Y 476.673,Z 393.926,A -85,B 0,C 180,E1 -7304.516,E2 -7304.516} C_VEL
LIN {X 0,Y 474.477,Z 379.829,A -85,B 0,C 180,E1 -7305.039,E2 -7305.039} C_VEL
LIN {X 0,Y 473.829,Z 376.006,A -85,B 0,C 180,E1 -7305.161,E2 -7305.161} C_VEL
LIN {X 0,Y 473.922,Z 369.67,A -85,B 0,C 180,E1 -7308.361,E2 -7308.361} C_VEL
LIN {X 0,Y 474.037,Z 363.167,A -85,B 0,C 180,E1 -7311.755,E2 -7311.755} C_VEL
LIN {X 0,Y 474.179,Z 358.034,A -85,B 0,C 180,E1 -7314.519,E2 -7314.519} C_VEL
LIN {X 0,Y 474.41,Z 352.95,A -85,B 0,C 180,E1 -7317.338,E2 -7317.338} C_VEL
LIN {X 0,Y 474.586,Z 347.926,A -85,B 0,C 180,E1 -7320.231,E2 -7320.231} C_VEL
LIN {X 0,Y 474.835,Z 343.021,A -85,B 0,C 180,E1 -7323.205,E2 -7323.205} C_VEL
LIN {X 0,Y 475.083,Z 338.186,A -85,B 0,C 180,E1 -7326.28,E2 -7326.28} C_VEL
LIN {X 0,Y 475.304,Z 333.477,A -85,B 0,C 180,E1 -7329.48,E2 -7329.48} C_VEL
LIN {X 0,Y 475.427,Z 329.548,A -85,B 0,C 180,E1 -7332.343,E2 -7332.343} C_VEL
LIN {X 0,Y 475.106,Z 326.523,A -85,B 0,C 180,E1 -7334.761,E2 -7334.761} C_VEL
LIN {X 0,Y 474.63,Z 323.048,A -85,B 0,C 180,E1 -7337.762,E2 -7337.762} C_VEL
LIN {X 0,Y 474.646,Z 322.863,A -85,B 0,C 180,E1 -7340.454,E2 -7340.454} C_VEL
LIN {X 0,Y 474.59,Z 322.87,A -85,B 0,C 180,E1 -7343.676,E2 -7343.676} C_VEL
LIN {X 0,Y 474.643,Z 322.857,A -85,B 0,C 180,E1 -7346.78,E2 -7346.78} C_VEL
LIN {X 0,Y 474.606,Z 322.868,A -85,B 0,C 180,E1 -7349.769,E2 -7349.769} C_VEL
LIN {X 0,Y 474.698,Z 322.85,A -85,B 0,C 180,E1 -7352.679,E2 -7352.679} C_VEL
LIN {X 0,Y 474.641,Z 322.862,A -85,B 0,C 180,E1 -7355.506,E2 -7355.506} C_VEL
LIN {X 0,Y 474.67,Z 322.855,A -85,B 0,C 180,E1 -7359.185,E2 -7359.185} C_VEL
LIN {X 0,Y 474.646,Z 322.861,A -85,B 0,C 180,E1 -7361.883,E2 -7361.883} C_VEL
LIN {X 0,Y 474.7,Z 322.85,A -85,B 0,C 180,E1 -7364.544,E2 -7364.544} C_VEL
LIN {X 0,Y 474.704,Z 322.851,A -85,B 0,C 180,E1 -7368.037,E2 -7368.037} C_VEL
LIN {X 0,Y 474.728,Z 322.853,A -85,B 0,C 180,E1 -7371.486,E2 -7371.486} C_VEL
LIN {X 0,Y 474.77,Z 322.841,A -85,B 0,C 180,E1 -7374.052,E2 -7374.052} C_VEL
LIN {X 0,Y 474.893,Z 322.831,A -85,B 0,C 180,E1 -7377.455,E2 -7377.455} C_VEL
LIN {X 0,Y 474.911,Z 322.824,A -85,B 0,C 180,E1 -7380,E2 -7380} C_VEL
LIN {X 0,Y 474.893,Z 322.827,A -85,B 0,C 180,E1 -7382.544,E2 -7382.544} C_VEL
LIN {X 0,Y 474.77,Z 322.841,A -85,B 0,C 180,E1 -7385.947,E2 -7385.947} C_VEL
LIN {X 0,Y 474.726,Z 322.849,A -85,B 0,C 180,E1 -7388.513,E2 -7388.513} C_VEL
LIN {X 0,Y 474.702,Z 322.849,A -85,B 0,C 180,E1 -7391.962,E2 -7391.962} C_VEL
LIN {X 0,Y 474.698,Z 322.851,A -85,B 0,C 180,E1 -7395.455,E2 -7395.455} C_VEL
LIN {X 0,Y 474.663,Z 322.859,A -85,B 0,C 180,E1 -7399.01,E2 -7399.01} C_VEL
LIN {X 0,Y 474.586,Z 322.864,A -85,B 0,C 180,E1 -7401.728,E2 -7401.728} C_VEL
LIN {X 0,Y 474.654,Z 322.862,A -85,B 0,C 180,E1 -7404.493,E2 -7404.493} C_VEL
LIN {X 0,Y 474.678,Z 322.853,A -85,B 0,C 180,E1 -7407.334,E2 -7407.334} C_VEL
LIN {X 0,Y 474.602,Z 322.865,A -85,B 0,C 180,E1 -7410.81,E2 -7410.81} C_VEL
LIN {X 0,Y 474.635,Z 322.861,A -85,B 0,C 180,E1 -7413.984,E2 -7413.984} C_VEL
LIN {X 0,Y 474.571,Z 322.867,A -85,B 0,C 180,E1 -7416.899,E2 -7416.899} C_VEL
LIN {X 0,Y 474.647,Z 322.858,A -85,B 0,C 180,E1 -7419.651,E2 -7419.651} C_VEL
LIN {X 0,Y 474.648,Z 322.857,A -85,B 0,C 180,E1 -7422.93,E2 -7422.93} C_VEL
LIN {X 0,Y 474.605,Z 322.867,A -85,B 0,C 180,E1 -7425.895,E2 -7425.895} C_VEL
LIN {X 0,Y 474.637,Z 322.857,A -85,B 0,C 180,E1 -7429.039,E2 -7429.039} C_VEL
LIN {X 0,Y 474.613,Z 322.866,A -85,B 0,C 180,E1 -7431.703,E2 -7431.703} C_VEL
LIN {X 0,Y 474.625,Z 322.859,A -85,B 0,C 180,E1 -7434.726,E2 -7434.726} C_VEL
LIN {X 0,Y 474.634,Z 322.866,A -85,B 0,C 180,E1 -7437.788,E2 -7437.788} C_VEL
LIN {X 0,Y 474.62,Z 322.86,A -85,B 0,C 180,E1 -7440.884,E2 -7440.884} C_VEL
LIN {X 0,Y 474.664,Z 322.863,A -85,B 0,C 180,E1 -7443.629,E2 -7443.629} C_VEL
LIN {X 0,Y 474.632,Z 322.858,A -85,B 0,C 180,E1 -7446.641,E2 -7446.641} C_VEL
LIN {X 0,Y 474.653,Z 322.857,A -85,B 0,C 180,E1 -7450.09,E2 -7450.09} C_VEL
LIN {X 0,Y 474.652,Z 322.862,A -85,B 0,C 180,E1 -7451.659,E2 -7451.659} C_VEL
LIN {X 0,Y 473.989,Z 322.943,A -85,B 0,C 180,E1 -7452.368,E2 -7452.368} C_VEL
LIN {X 0,Y 471.14,Z 323.301,A -85,B 0,C 180,E1 -7453.519,E2 -7453.519} C_VEL
LIN {X 0,Y 468.726,Z 323.603,A -85,B 0,C 180,E1 -7454.447,E2 -7454.447} C_VEL
LIN {X 0,Y 467.684,Z 323.731,A -85,B 0,C 180,E1 -7455.165,E2 -7455.165} C_VEL
LIN {X 0,Y 467.597,Z 323.74,A -85,B 0,C 180,E1 -7455.407,E2 -7455.407} C_VEL
LIN {X 0,Y 467.65,Z 323.732,A -85,B 0,C 180,E1 -7458.734,E2 -7458.734} C_VEL
LIN {X 0,Y 467.745,Z 323.72,A -85,B 0,C 180,E1 -7462.228,E2 -7462.228} C_VEL
LIN {X 0,Y 467.723,Z 323.725,A -85,B 0,C 180,E1 -7464.827,E2 -7464.827} C_VEL
LIN {X 0,Y 467.857,Z 323.708,A -85,B 0,C 180,E1 -7467.417,E2 -7467.417} C_VEL
LIN {X 0,Y 467.88,Z 323.703,A -85,B 0,C 180,E1 -7470,E2 -7470} C_VEL
LIN {X 0,Y 467.857,Z 323.708,A -85,B 0,C 180,E1 -7472.583,E2 -7472.583} C_VEL
LIN {X 0,Y 467.743,Z 323.72,A -85,B 0,C 180,E1 -7476.037,E2 -7476.037} C_VEL
LIN {X 0,Y 467.679,Z 323.732,A -85,B 0,C 180,E1 -7478.643,E2 -7478.643} C_VEL
LIN {X 0,Y 467.652,Z 323.731,A -85,B 0,C 180,E1 -7482.145,E2 -7482.145} C_VEL
LIN {X 0,Y 467.636,Z 323.733,A -85,B 0,C 180,E1 -7485.695,E2 -7485.695} C_VEL
LIN {X 0,Y 467.614,Z 323.74,A -85,B 0,C 180,E1 -7488.765,E2 -7488.765} C_VEL
LIN {X 0,Y 467.576,Z 323.737,A -85,B 0,C 180,E1 -7491.268,E2 -7491.268} C_VEL
LIN {X 0,Y 467.568,Z 323.74,A -85,B 0,C 180,E1 -7493.943,E2 -7493.943} C_VEL
LIN {X 0,Y 467.624,Z 323.734,A -85,B 0,C 180,E1 -7496.8,E2 -7496.8} C_VEL
LIN {X 0,Y 467.551,Z 323.742,A -85,B 0,C 180,E1 -7499.738,E2 -7499.738} C_VEL
LIN {X 0,Y 467.58,Z 323.738,A -85,B 0,C 180,E1 -7502.758,E2 -7502.758} C_VEL
LIN {X 0,Y 467.552,Z 323.745,A -85,B 0,C 180,E1 -7505.89,E2 -7505.89} C_VEL
LIN {X 0,Y 467.596,Z 323.735,A -85,B 0,C 180,E1 -7509.143,E2 -7509.143} C_VEL
LIN {X 0,Y 467.582,Z 323.738,A -85,B 0,C 180,E1 -7512.567,E2 -7512.567} C_VEL
LIN {X 0,Y 467.567,Z 323.738,A -85,B 0,C 180,E1 -7515.053,E2 -7515.053} C_VEL
LIN {X 0,Y 467.621,Z 323.734,A -85,B 0,C 180,E1 -7517.444,E2 -7517.444} C_VEL
LIN {X 0,Y 467.596,Z 323.735,A -85,B 0,C 180,E1 -7520.857,E2 -7520.857} C_VEL
LIN {X 0,Y 467.556,Z 323.741,A -85,B 0,C 180,E1 -7524.261,E2 -7524.261} C_VEL
LIN {X 0,Y 467.579,Z 323.741,A -85,B 0,C 180,E1 -7527.321,E2 -7527.321} C_VEL
LIN {X 0,Y 467.567,Z 323.738,A -85,B 0,C 180,E1 -7530.668,E2 -7530.668} C_VEL
LIN {X 0,Y 467.614,Z 323.737,A -85,B 0,C 180,E1 -7533.2,E2 -7533.2} C_VEL
LIN {X 0,Y 467.59,Z 323.735,A -85,B 0,C 180,E1 -7536.469,E2 -7536.469} C_VEL
LIN {X 0,Y 467.622,Z 323.734,A -85,B 0,C 180,E1 -7539.778,E2 -7539.778} C_VEL
LIN {X 0,Y 467.607,Z 323.734,A -85,B 0,C 180,E1 -7542.507,E2 -7542.507} C_VEL
LIN {X 0,Y 467.605,Z 323.742,A -85,B 0,C 180,E1 -7545.197,E2 -7545.197} C_VEL
LIN {X 0,Y 467.654,Z 323.728,A -85,B 0,C 180,E1 -7547.855,E2 -7547.855} C_VEL
LIN {X 0,Y 467.68,Z 323.728,A -85,B 0,C 180,E1 -7551.358,E2 -7551.358} C_VEL
LIN {X 0,Y 467.734,Z 323.717,A -85,B 0,C 180,E1 -7553.963,E2 -7553.963} C_VEL
LIN {X 0,Y 467.859,Z 323.704,A -85,B 0,C 180,E1 -7557.418,E2 -7557.418} C_VEL
LIN {X 0,Y 467.881,Z 323.699,A -85,B 0,C 180,E1 -7560,E2 -7560} C_VEL
LIN {X 0,Y 467.859,Z 323.708,A -85,B 0,C 180,E1 -7562.583,E2 -7562.583} C_VEL
LIN {X 0,Y 467.735,Z 323.718,A -85,B 0,C 180,E1 -7566.038,E2 -7566.038} C_VEL
LIN {X 0,Y 467.681,Z 323.732,A -85,B 0,C 180,E1 -7568.643,E2 -7568.643} C_VEL
LIN {X 0,Y 467.656,Z 323.73,A -85,B 0,C 180,E1 -7572.146,E2 -7572.146} C_VEL
LIN {X 0,Y 467.639,Z 323.73,A -85,B 0,C 180,E1 -7575.695,E2 -7575.695} C_VEL
LIN {X 0,Y 467.613,Z 323.736,A -85,B 0,C 180,E1 -7578.763,E2 -7578.763} C_VEL
LIN {X 0,Y 467.58,Z 323.737,A -85,B 0,C 180,E1 -7581.269,E2 -7581.269} C_VEL
LIN {X 0,Y 467.563,Z 323.743,A -85,B 0,C 180,E1 -7583.944,E2 -7583.944} C_VEL
LIN {X 0,Y 467.613,Z 323.734,A -85,B 0,C 180,E1 -7586.801,E2 -7586.801} C_VEL
LIN {X 0,Y 467.554,Z 323.743,A -85,B 0,C 180,E1 -7589.739,E2 -7589.739} C_VEL
LIN {X 0,Y 467.584,Z 323.737,A -85,B 0,C 180,E1 -7592.759,E2 -7592.759} C_VEL
LIN {X 0,Y 467.554,Z 323.747,A -85,B 0,C 180,E1 -7595.89,E2 -7595.89} C_VEL
LIN {X 0,Y 467.583,Z 323.742,A -85,B 0,C 180,E1 -7599.145,E2 -7599.145} C_VEL
LIN {X 0,Y 467.577,Z 323.745,A -85,B 0,C 180,E1 -7601.403,E2 -7601.403} C_VEL
LIN {X 0,Y 467.682,Z 324.635,A -85,B 0,C 180,E1 -7602.58,E2 -7602.58} C_VEL
LIN {X 0,Y 468.285,Z 328.7,A -85,B 0,C 180,E1 -7606.086,E2 -7606.086} C_VEL
LIN {X 0,Y 468.407,Z 332.029,A -85,B 0,C 180,E1 -7608.687,E2 -7608.687} C_VEL
LIN {X 0,Y 468.186,Z 336.677,A -85,B 0,C 180,E1 -7612.015,E2 -7612.015} C_VEL
LIN {X 0,Y 467.944,Z 341.436,A -85,B 0,C 180,E1 -7615.2,E2 -7615.2} C_VEL
LIN {X 0,Y 467.688,Z 346.296,A -85,B 0,C 180,E1 -7618.268,E2 -7618.268} C_VEL
LIN {X 0,Y 467.429,Z 351.253,A -85,B 0,C 180,E1 -7621.241,E2 -7621.241} C_VEL
LIN {X 0,Y 467.204,Z 356.278,A -85,B 0,C 180,E1 -7624.136,E2 -7624.136} C_VEL
LIN {X 0,Y 467.048,Z 361.365,A -85,B 0,C 180,E1 -7626.968,E2 -7626.968} C_VEL
LIN {X 0,Y 466.907,Z 366.532,A -85,B 0,C 180,E1 -7629.745,E2 -7629.745} C_VEL
LIN {X 0,Y 466.791,Z 371.709,A -85,B 0,C 180,E1 -7632.475,E2 -7632.475} C_VEL
LIN {X 0,Y 466.728,Z 376.085,A -85,B 0,C 180,E1 -7634.631,E2 -7634.631} C_VEL
LIN {X 0,Y 468.48,Z 386.014,A -85,B 0,C 180,E1 -7634.951,E2 -7634.951} C_VEL
LIN {X 0,Y 469.962,Z 396.314,A -85,B 0,C 180,E1 -7635.383,E2 -7635.383} C_VEL
LIN {X 0,Y 469.582,Z 406.398,A -85,B 0,C 180,E1 -7635.869,E2 -7635.869} C_VEL
LIN {X 0,Y 469.187,Z 416.16,A -85,B 0,C 180,E1 -7636.465,E2 -7636.465} C_VEL
LIN {X 0,Y 468.649,Z 426.686,A -85,B 0,C 180,E1 -7637.258,E2 -7637.258} C_VEL
LIN {X 0,Y 468.204,Z 437.736,A -85,B 0,C 180,E1 -7638.309,E2 -7638.309} C_VEL
LIN {X 0,Y 467.762,Z 446.878,A -85,B 0,C 180,E1 -7639.394,E2 -7639.394} C_VEL
LIN {X 0,Y 467.471,Z 453.081,A -85,B 0,C 180,E1 -7640.263,E2 -7640.263} C_VEL
LIN {X 0,Y 467.206,Z 459.619,A -85,B 0,C 180,E1 -7641.348,E2 -7641.348} C_VEL
LIN {X 0,Y 467.01,Z 464.121,A -85,B 0,C 180,E1 -7642.216,E2 -7642.216} C_VEL
LIN {X 0,Y 466.808,Z 469.718,A -85,B 0,C 180,E1 -7643.547,E2 -7643.547} C_VEL
LIN {X 0,Y 466.742,Z 473.933,A -85,B 0,C 180,E1 -7644.817,E2 -7644.817} C_VEL
LIN {X 0,Y 466.649,Z 476.296,A -85,B 0,C 180,E1 -7645.681,E2 -7645.681} C_VEL
LIN {X 0,Y 466.69,Z 478.094,A -85,B 0,C 180,E1 -7646.547,E2 -7646.547} C_VEL
LIN {X 0,Y 466.608,Z 480.534,A -85,B 0,C 180,E1 -7648.274,E2 -7648.274} C_VEL
LIN {X 0,Y 466.619,Z 481.122,A -85,B 0,C 180,E1 -7649.137,E2 -7649.137} C_VEL
LIN {X 0,Y 466.619,Z 481.122,A -85,B 0,C 180,E1 -7650.863,E2 -7650.863} C_VEL
LIN {X 0,Y 466.608,Z 480.534,A -85,B 0,C 180,E1 -7651.726,E2 -7651.726} C_VEL
LIN {X 0,Y 466.69,Z 478.094,A -85,B 0,C 180,E1 -7653.453,E2 -7653.453} C_VEL
LIN {X 0,Y 466.694,Z 475.148,A -85,B 0,C 180,E1 -7654.751,E2 -7654.751} C_VEL
LIN {X 0,Y 466.762,Z 471.163,A -85,B 0,C 180,E1 -7656.05,E2 -7656.05} C_VEL
LIN {X 0,Y 466.943,Z 466.036,A -85,B 0,C 180,E1 -7657.35,E2 -7657.35} C_VEL
LIN {X 0,Y 467.154,Z 460.775,A -85,B 0,C 180,E1 -7658.435,E2 -7658.435} C_VEL
LIN {X 0,Y 467.384,Z 454.456,A -85,B 0,C 180,E1 -7659.521,E2 -7659.521} C_VEL
LIN {X 0,Y 467.645,Z 448.504,A -85,B 0,C 180,E1 -7660.39,E2 -7660.39} C_VEL
LIN {X 0,Y 468.059,Z 441.577,A -85,B 0,C 180,E1 -7661.256,E2 -7661.256} C_VEL
LIN {X 0,Y 468.434,Z 433.395,A -85,B 0,C 180,E1 -7662.125,E2 -7662.125} C_VEL
LIN {X 0,Y 468.715,Z 425.114,A -85,B 0,C 180,E1 -7662.868,E2 -7662.868} C_VEL
LIN {X 0,Y 469.131,Z 416.158,A -85,B 0,C 180,E1 -7663.537,E2 -7663.537} C_VEL
LIN {X 0,Y 469.576,Z 406.398,A -85,B 0,C 180,E1 -7664.131,E2 -7664.131} C_VEL
LIN {X 0,Y 469.933,Z 397.602,A -85,B 0,C 180,E1 -7664.562,E2 -7664.562} C_VEL
LIN {X 0,Y 468.765,Z 388.04,A -85,B 0,C 180,E1 -7664.975,E2 -7664.975} C_VEL
LIN {X 0,Y 466.983,Z 377.617,A -85,B 0,C 180,E1 -7665.328,E2 -7665.328} C_VEL
LIN {X 0,Y 466.701,Z 375.844,A -85,B 0,C 180,E1 -7665.399,E2 -7665.399} C_VEL
LIN {X 0,Y 466.854,Z 369.85,A -85,B 0,C 180,E1 -7668.485,E2 -7668.485} C_VEL
LIN {X 0,Y 466.937,Z 364.784,A -85,B 0,C 180,E1 -7671.176,E2 -7671.176} C_VEL
LIN {X 0,Y 467.06,Z 359.659,A -85,B 0,C 180,E1 -7673.971,E2 -7673.971} C_VEL
LIN {X 0,Y 467.293,Z 354.585,A -85,B 0,C 180,E1 -7676.82,E2 -7676.82} C_VEL
LIN {X 0,Y 467.488,Z 349.579,A -85,B 0,C 180,E1 -7679.743,E2 -7679.743} C_VEL
LIN {X 0,Y 467.78,Z 344.656,A -85,B 0,C 180,E1 -7682.743,E2 -7682.743} C_VEL
LIN {X 0,Y 468.013,Z 339.823,A -85,B 0,C 180,E1 -7685.849,E2 -7685.849} C_VEL
LIN {X 0,Y 468.234,Z 335.097,A -85,B 0,C 180,E1 -7689.08,E2 -7689.08} C_VEL
LIN {X 0,Y 468.4,Z 331.901,A -85,B 0,C 180,E1 -7691.391,E2 -7691.391} C_VEL
LIN {X 0,Y 468.285,Z 328.674,A -85,B 0,C 180,E1 -7693.914,E2 -7693.914} C_VEL
LIN {X 0,Y 467.691,Z 324.597,A -85,B 0,C 180,E1 -7697.451,E2 -7697.451} C_VEL
LIN {X 0,Y 467.579,Z 323.743,A -85,B 0,C 180,E1 -7698.723,E2 -7698.723} C_VEL
LIN {X 0,Y 467.566,Z 323.746,A -85,B 0,C 180,E1 -7701.955,E2 -7701.955} C_VEL
LIN {X 0,Y 467.565,Z 323.743,A -85,B 0,C 180,E1 -7705.167,E2 -7705.167} C_VEL
LIN {X 0,Y 467.583,Z 323.74,A -85,B 0,C 180,E1 -7708.259,E2 -7708.259} C_VEL
LIN {X 0,Y 467.577,Z 323.738,A -85,B 0,C 180,E1 -7711.25,E2 -7711.25} C_VEL
LIN {X 0,Y 467.597,Z 323.738,A -85,B 0,C 180,E1 -7714.159,E2 -7714.159} C_VEL
LIN {X 0,Y 467.576,Z 323.738,A -85,B 0,C 180,E1 -7716.995,E2 -7716.995} C_VEL
LIN {X 0,Y 467.622,Z 323.738,A -85,B 0,C 180,E1 -7719.777,E2 -7719.777} C_VEL
LIN {X 0,Y 467.598,Z 323.734,A -85,B 0,C 180,E1 -7722.506,E2 -7722.506} C_VEL
LIN {X 0,Y 467.609,Z 323.737,A -85,B 0,C 180,E1 -7725.196,E2 -7725.196} C_VEL
LIN {X 0,Y 467.656,Z 323.73,A -85,B 0,C 180,E1 -7727.854,E2 -7727.854} C_VEL
LIN {X 0,Y 467.681,Z 323.732,A -85,B 0,C 180,E1 -7731.357,E2 -7731.357} C_VEL
LIN {X 0,Y 467.735,Z 323.718,A -85,B 0,C 180,E1 -7733.962,E2 -7733.962} C_VEL
LIN {X 0,Y 467.859,Z 323.708,A -85,B 0,C 180,E1 -7737.417,E2 -7737.417} C_VEL
LIN {X 0,Y 467.881,Z 323.699,A -85,B 0,C 180,E1 -7740,E2 -7740} C_VEL
LIN {X 0,Y 467.859,Z 323.704,A -85,B 0,C 180,E1 -7742.582,E2 -7742.582} C_VEL
LIN {X 0,Y 467.734,Z 323.717,A -85,B 0,C 180,E1 -7746.037,E2 -7746.037} C_VEL
LIN {X 0,Y 467.68,Z 323.728,A -85,B 0,C 180,E1 -7748.642,E2 -7748.642} C_VEL
LIN {X 0,Y 467.654,Z 323.728,A -85,B 0,C 180,E1 -7752.145,E2 -7752.145} C_VEL
LIN {X 0,Y 467.637,Z 323.73,A -85,B 0,C 180,E1 -7755.695,E2 -7755.695} C_VEL
LIN {X 0,Y 467.616,Z 323.74,A -85,B 0,C 180,E1 -7758.764,E2 -7758.764} C_VEL
LIN {X 0,Y 467.578,Z 323.738,A -85,B 0,C 180,E1 -7761.268,E2 -7761.268} C_VEL
LIN {X 0,Y 467.569,Z 323.739,A -85,B 0,C 180,E1 -7763.943,E2 -7763.943} C_VEL
LIN {X 0,Y 467.614,Z 323.737,A -85,B 0,C 180,E1 -7766.8,E2 -7766.8} C_VEL
LIN {X 0,Y 467.551,Z 323.741,A -85,B 0,C 180,E1 -7769.738,E2 -7769.738} C_VEL
LIN {X 0,Y 467.581,Z 323.74,A -85,B 0,C 180,E1 -7772.758,E2 -7772.758} C_VEL
LIN {X 0,Y 467.552,Z 323.743,A -85,B 0,C 180,E1 -7775.889,E2 -7775.889} C_VEL
LIN {X 0,Y 467.596,Z 323.735,A -85,B 0,C 180,E1 -7779.143,E2 -7779.143} C_VEL
LIN {X 0,Y 467.616,Z 323.735,A -85,B 0,C 180,E1 -7782.571,E2 -7782.571} C_VEL
LIN {X 0,Y 467.567,Z 323.738,A -85,B 0,C 180,E1 -7785.053,E2 -7785.053} C_VEL
LIN {X 0,Y 467.585,Z 323.737,A -85,B 0,C 180,E1 -7787.44,E2 -7787.44} C_VEL
LIN {X 0,Y 467.596,Z 323.735,A -85,B 0,C 180,E1 -7790.857,E2 -7790.857} C_VEL
LIN {X 0,Y 467.558,Z 323.742,A -85,B 0,C 180,E1 -7794.26,E2 -7794.26} C_VEL
LIN {X 0,Y 467.579,Z 323.739,A -85,B 0,C 180,E1 -7797.321,E2 -7797.321} C_VEL
LIN {X 0,Y 467.566,Z 323.738,A -85,B 0,C 180,E1 -7800.667,E2 -7800.667} C_VEL
LIN {X 0,Y 467.624,Z 323.734,A -85,B 0,C 180,E1 -7803.2,E2 -7803.2} C_VEL
LIN {X 0,Y 467.589,Z 323.736,A -85,B 0,C 180,E1 -7806.468,E2 -7806.468} C_VEL
LIN {X 0,Y 467.62,Z 323.736,A -85,B 0,C 180,E1 -7809.777,E2 -7809.777} C_VEL
LIN {X 0,Y 467.605,Z 323.736,A -85,B 0,C 180,E1 -7812.507,E2 -7812.507} C_VEL
LIN {X 0,Y 467.597,Z 323.74,A -85,B 0,C 180,E1 -7815.407,E2 -7815.407} C_VEL
LIN {X 0,Y 466.925,Z 323.823,A -85,B 0,C 180,E1 -7816.127,E2 -7816.127} C_VEL
LIN {X 0,Y 464.081,Z 324.181,A -85,B 0,C 180,E1 -7817.295,E2 -7817.295} C_VEL
LIN {X 0,Y 461.683,Z 324.476,A -85,B 0,C 180,E1 -7818.237,E2 -7818.237} C_VEL
LIN {X 0,Y 460.656,Z 324.605,A -85,B 0,C 180,E1 -7818.965,E2 -7818.965} C_VEL
LIN {X 0,Y 460.574,Z 324.614,A -85,B 0,C 180,E1 -7819.211,E2 -7819.211} C_VEL
LIN {X 0,Y 460.716,Z 324.596,A -85,B 0,C 180,E1 -7822.538,E2 -7822.538} C_VEL
LIN {X 0,Y 460.696,Z 324.6,A -85,B 0,C 180,E1 -7824.748,E2 -7824.748} C_VEL
LIN {X 0,Y 460.822,Z 324.585,A -85,B 0,C 180,E1 -7827.378,E2 -7827.378} C_VEL
LIN {X 0,Y 460.85,Z 324.579,A -85,B 0,C 180,E1 -7830,E2 -7830} C_VEL
LIN {X 0,Y 460.822,Z 324.585,A -85,B 0,C 180,E1 -7832.622,E2 -7832.622} C_VEL
LIN {X 0,Y 460.708,Z 324.597,A -85,B 0,C 180,E1 -7836.13,E2 -7836.13} C_VEL
LIN {X 0,Y 460.626,Z 324.611,A -85,B 0,C 180,E1 -7838.776,E2 -7838.776} C_VEL
LIN {X 0,Y 460.61,Z 324.61,A -85,B 0,C 180,E1 -7842.445,E2 -7842.445} C_VEL
LIN {X 0,Y 460.596,Z 324.611,A -85,B 0,C 180,E1 -7845.998,E2 -7845.998} C_VEL
LIN {X 0,Y 460.568,Z 324.616,A -85,B 0,C 180,E1 -7848.902,E2 -7848.902} C_VEL
LIN {X 0,Y 460.512,Z 324.617,A -85,B 0,C 180,E1 -7851.486,E2 -7851.486} C_VEL
LIN {X 0,Y 460.538,Z 324.621,A -85,B 0,C 180,E1 -7854.332,E2 -7854.332} C_VEL
LIN {X 0,Y 460.58,Z 324.609,A -85,B 0,C 180,E1 -7857.243,E2 -7857.243} C_VEL
LIN {X 0,Y 460.507,Z 324.626,A -85,B 0,C 180,E1 -7860.24,E2 -7860.24} C_VEL
LIN {X 0,Y 460.526,Z 324.616,A -85,B 0,C 180,E1 -7863.325,E2 -7863.325} C_VEL
LIN {X 0,Y 460.475,Z 324.625,A -85,B 0,C 180,E1 -7866.529,E2 -7866.529} C_VEL
LIN {X 0,Y 460.571,Z 324.615,A -85,B 0,C 180,E1 -7869.858,E2 -7869.858} C_VEL
LIN {X 0,Y 460.509,Z 324.618,A -85,B 0,C 180,E1 -7872.901,E2 -7872.901} C_VEL
LIN {X 0,Y 460.52,Z 324.623,A -85,B 0,C 180,E1 -7875.829,E2 -7875.829} C_VEL
LIN {X 0,Y 460.54,Z 324.614,A -85,B 0,C 180,E1 -7878.99,E2 -7878.99} C_VEL
LIN {X 0,Y 460.536,Z 324.616,A -85,B 0,C 180,E1 -7881.269,E2 -7881.269} C_VEL
LIN {X 0,Y 460.507,Z 324.618,A -85,B 0,C 180,E1 -7884.555,E2 -7884.555} C_VEL
LIN {X 0,Y 460.529,Z 324.622,A -85,B 0,C 180,E1 -7887.716,E2 -7887.716} C_VEL
LIN {X 0,Y 460.537,Z 324.615,A -85,B 0,C 180,E1 -7890.769,E2 -7890.769} C_VEL
LIN {X 0,Y 460.561,Z 324.615,A -85,B 0,C 180,E1 -7893.735,E2 -7893.735} C_VEL
LIN {X 0,Y 460.543,Z 324.614,A -85,B 0,C 180,E1 -7896.624,E2 -7896.624} C_VEL
LIN {X 0,Y 460.55,Z 324.619,A -85,B 0,C 180,E1 -7899.453,E2 -7899.453} C_VEL
LIN {X 0,Y 460.557,Z 324.612,A -85,B 0,C 180,E1 -7902.231,E2 -7902.231} C_VEL
LIN {X 0,Y 460.564,Z 324.616,A -85,B 0,C 180,E1 -7904.965,E2 -7904.965} C_VEL
LIN {X 0,Y 460.609,Z 324.607,A -85,B 0,C 180,E1 -7908.56,E2 -7908.56} C_VEL
LIN {X 0,Y 460.694,Z 324.595,A -85,B 0,C 180,E1 -7912.109,E2 -7912.109} C_VEL
LIN {X 0,Y 460.693,Z 324.6,A -85,B 0,C 180,E1 -7914.749,E2 -7914.749} C_VEL
LIN {X 0,Y 460.824,Z 324.58,A -85,B 0,C 180,E1 -7917.378,E2 -7917.378} C_VEL
LIN {X 0,Y 460.852,Z 324.575,A -85,B 0,C 180,E1 -7920,E2 -7920} C_VEL
LIN {X 0,Y 460.823,Z 324.585,A -85,B 0,C 180,E1 -7922.623,E2 -7922.623} C_VEL
LIN {X 0,Y 460.701,Z 324.595,A -85,B 0,C 180,E1 -7926.13,E2 -7926.13} C_VEL
LIN {X 0,Y 460.628,Z 324.608,A -85,B 0,C 180,E1 -7928.777,E2 -7928.777} C_VEL
LIN {X 0,Y 460.613,Z 324.612,A -85,B 0,C 180,E1 -7932.445,E2 -7932.445} C_VEL
LIN {X 0,Y 460.6,Z 324.609,A -85,B 0,C 180,E1 -7935.998,E2 -7935.998} C_VEL
LIN {X 0,Y 460.568,Z 324.611,A -85,B 0,C 180,E1 -7939.616,E2 -7939.616} C_VEL
LIN {X 0,Y 460.511,Z 324.623,A -85,B 0,C 180,E1 -7942.429,E2 -7942.429} C_VEL
LIN {X 0,Y 460.553,Z 324.615,A -85,B 0,C 180,E1 -7945.798,E2 -7945.798} C_VEL
LIN {X 0,Y 460.553,Z 324.619,A -85,B 0,C 180,E1 -7948.233,E2 -7948.233} C_VEL
LIN {X 0,Y 460.521,Z 324.616,A -85,B 0,C 180,E1 -7951.283,E2 -7951.283} C_VEL
LIN {X 0,Y 460.532,Z 324.618,A -85,B 0,C 180,E1 -7954.506,E2 -7954.506} C_VEL
LIN {X 0,Y 460.502,Z 324.626,A -85,B 0,C 180,E1 -7957.624,E2 -7957.624} C_VEL
LIN {X 0,Y 460.543,Z 324.621,A -85,B 0,C 180,E1 -7960.27,E2 -7960.27} C_VEL
LIN {X 0,Y 460.546,Z 324.762,A -85,B 0,C 180,E1 -7961.605,E2 -7961.605} C_VEL
LIN {X 0,Y 460.999,Z 327.995,A -85,B 0,C 180,E1 -7964.53,E2 -7964.53} C_VEL
LIN {X 0,Y 461.367,Z 330.921,A -85,B 0,C 180,E1 -7966.986,E2 -7966.986} C_VEL
LIN {X 0,Y 461.297,Z 334.364,A -85,B 0,C 180,E1 -7969.621,E2 -7969.621} C_VEL
LIN {X 0,Y 461.143,Z 338.275,A -85,B 0,C 180,E1 -7972.438,E2 -7972.438} C_VEL
LIN {X 0,Y 460.877,Z 343.062,A -85,B 0,C 180,E1 -7975.652,E2 -7975.652} C_VEL
LIN {X 0,Y 460.581,Z 347.911,A -85,B 0,C 180,E1 -7978.748,E2 -7978.748} C_VEL
LIN {X 0,Y 460.321,Z 352.873,A -85,B 0,C 180,E1 -7981.752,E2 -7981.752} C_VEL
LIN {X 0,Y 460.129,Z 357.892,A -85,B 0,C 180,E1 -7984.68,E2 -7984.68} C_VEL
LIN {X 0,Y 459.908,Z 362.971,A -85,B 0,C 180,E1 -7987.54,E2 -7987.54} C_VEL
LIN {X 0,Y 459.79,Z 368.11,A -85,B 0,C 180,E1 -7990.35,E2 -7990.35} C_VEL
LIN {X 0,Y 459.684,Z 373.286,A -85,B 0,C 180,E1 -7993.113,E2 -7993.113} C_VEL
LIN {X 0,Y 459.64,Z 375.713,A -85,B 0,C 180,E1 -7994.373,E2 -7994.373} C_VEL
LIN {X 0,Y 461.893,Z 388.782,A -85,B 0,C 180,E1 -7994.827,E2 -7994.827} C_VEL
LIN {X 0,Y 463.063,Z 397.406,A -85,B 0,C 180,E1 -7995.217,E2 -7995.217} C_VEL
LIN {X 0,Y 462.589,Z 409.224,A -85,B 0,C 180,E1 -7995.819,E2 -7995.819} C_VEL
LIN {X 0,Y 462.023,Z 420.626,A -85,B 0,C 180,E1 -7996.587,E2 -7996.587} C_VEL
LIN {X 0,Y 461.607,Z 429.983,A -85,B 0,C 180,E1 -7997.377,E2 -7997.377} C_VEL
LIN {X 0,Y 461.246,Z 437.54,A -85,B 0,C 180,E1 -7998.13,E2 -7998.13} C_VEL
LIN {X 0,Y 460.751,Z 446.681,A -85,B 0,C 180,E1 -7999.231,E2 -7999.231} C_VEL
LIN {X 0,Y 460.458,Z 452.884,A -85,B 0,C 180,E1 -8000.113,E2 -8000.113} C_VEL
LIN {X 0,Y 460.154,Z 459.423,A -85,B 0,C 180,E1 -8001.215,E2 -8001.215} C_VEL
LIN {X 0,Y 459.95,Z 463.924,A -85,B 0,C 180,E1 -8002.096,E2 -8002.096} C_VEL
LIN {X 0,Y 459.748,Z 468.907,A -85,B 0,C 180,E1 -8003.273,E2 -8003.273} C_VEL
LIN {X 0,Y 459.656,Z 473.737,A -85,B 0,C 180,E1 -8004.736,E2 -8004.736} C_VEL
LIN {X 0,Y 459.567,Z 476.1,A -85,B 0,C 180,E1 -8005.615,E2 -8005.615} C_VEL
LIN {X 0,Y 459.585,Z 477.898,A -85,B 0,C 180,E1 -8006.493,E2 -8006.493} C_VEL
LIN {X 0,Y 459.521,Z 480.338,A -85,B 0,C 180,E1 -8008.247,E2 -8008.247} C_VEL
LIN {X 0,Y 459.522,Z 480.926,A -85,B 0,C 180,E1 -8009.124,E2 -8009.124} C_VEL
LIN {X 0,Y 459.522,Z 480.926,A -85,B 0,C 180,E1 -8010.876,E2 -8010.876} C_VEL
LIN {X 0,Y 459.521,Z 480.338,A -85,B 0,C 180,E1 -8011.753,E2 -8011.753} C_VEL
LIN {X 0,Y 459.585,Z 477.898,A -85,B 0,C 180,E1 -8013.507,E2 -8013.507} C_VEL
LIN {X 0,Y 459.621,Z 474.953,A -85,B 0,C 180,E1 -8014.824,E2 -8014.824} C_VEL
LIN {X 0,Y 459.671,Z 470.966,A -85,B 0,C 180,E1 -8016.144,E2 -8016.144} C_VEL
LIN {X 0,Y 459.865,Z 465.839,A -85,B 0,C 180,E1 -8017.464,E2 -8017.464} C_VEL
LIN {X 0,Y 460.116,Z 460.579,A -85,B 0,C 180,E1 -8018.565,E2 -8018.565} C_VEL
LIN {X 0,Y 460.37,Z 454.26,A -85,B 0,C 180,E1 -8019.667,E2 -8019.667} C_VEL
LIN {X 0,Y 460.628,Z 448.307,A -85,B 0,C 180,E1 -8020.55,E2 -8020.55} C_VEL
LIN {X 0,Y 461.056,Z 441.38,A -85,B 0,C 180,E1 -8021.429,E2 -8021.429} C_VEL
LIN {X 0,Y 461.454,Z 433.198,A -85,B 0,C 180,E1 -8022.311,E2 -8022.311} C_VEL
LIN {X 0,Y 461.782,Z 424.692,A -85,B 0,C 180,E1 -8023.083,E2 -8023.083} C_VEL
LIN {X 0,Y 462.228,Z 415.963,A -85,B 0,C 180,E1 -8023.743,E2 -8023.743} C_VEL
LIN {X 0,Y 462.693,Z 406.202,A -85,B 0,C 180,E1 -8024.346,E2 -8024.346} C_VEL
LIN {X 0,Y 463.059,Z 397.406,A -85,B 0,C 180,E1 -8024.784,E2 -8024.784} C_VEL
LIN {X 0,Y 461.577,Z 386.721,A -85,B 0,C 180,E1 -8025.25,E2 -8025.25} C_VEL
LIN {X 0,Y 459.64,Z 375.713,A -85,B 0,C 180,E1 -8025.627,E2 -8025.627} C_VEL
LIN {X 0,Y 459.77,Z 369.822,A -85,B 0,C 180,E1 -8028.724,E2 -8028.724} C_VEL
LIN {X 0,Y 459.883,Z 364.675,A -85,B 0,C 180,E1 -8031.517,E2 -8031.517} C_VEL
LIN {X 0,Y 460.015,Z 359.574,A -85,B 0,C 180,E1 -8034.362,E2 -8034.362} C_VEL
LIN {X 0,Y 460.3,Z 353.81,A -85,B 0,C 180,E1 -8037.679,E2 -8037.679} C_VEL
LIN {X 0,Y 460.496,Z 349.549,A -85,B 0,C 180,E1 -8040.241,E2 -8040.241} C_VEL
LIN {X 0,Y 460.747,Z 344.653,A -85,B 0,C 180,E1 -8043.307,E2 -8043.307} C_VEL
LIN {X 0,Y 460.978,Z 340.411,A -85,B 0,C 180,E1 -8046.096,E2 -8046.096} C_VEL
LIN {X 0,Y 461.204,Z 336.236,A -85,B 0,C 180,E1 -8048.998,E2 -8048.998} C_VEL
LIN {X 0,Y 461.382,Z 332.085,A -85,B 0,C 180,E1 -8052.084,E2 -8052.084} C_VEL
LIN {X 0,Y 461.165,Z 329.106,A -85,B 0,C 180,E1 -8054.509,E2 -8054.509} C_VEL
LIN {X 0,Y 460.626,Z 325.367,A -85,B 0,C 180,E1 -8057.83,E2 -8057.83} C_VEL
LIN {X 0,Y 460.546,Z 324.761,A -85,B 0,C 180,E1 -8058.395,E2 -8058.395} C_VEL
LIN {X 0,Y 460.527,Z 324.62,A -85,B 0,C 180,E1 -8061.267,E2 -8061.267} C_VEL
LIN {X 0,Y 460.511,Z 324.624,A -85,B 0,C 180,E1 -8064.554,E2 -8064.554} C_VEL
LIN {X 0,Y 460.532,Z 324.619,A -85,B 0,C 180,E1 -8067.715,E2 -8067.715} C_VEL
LIN {X 0,Y 460.54,Z 324.614,A -85,B 0,C 180,E1 -8070.769,E2 -8070.769} C_VEL
LIN {X 0,Y 460.556,Z 324.619,A -85,B 0,C 180,E1 -8073.734,E2 -8073.734} C_VEL
LIN {X 0,Y 460.545,Z 324.613,A -85,B 0,C 180,E1 -8076.623,E2 -8076.623} C_VEL
LIN {X 0,Y 460.551,Z 324.617,A -85,B 0,C 180,E1 -8079.452,E2 -8079.452} C_VEL
LIN {X 0,Y 460.549,Z 324.614,A -85,B 0,C 180,E1 -8082.229,E2 -8082.229} C_VEL
LIN {X 0,Y 460.567,Z 324.612,A -85,B 0,C 180,E1 -8084.964,E2 -8084.964} C_VEL
LIN {X 0,Y 460.611,Z 324.605,A -85,B 0,C 180,E1 -8088.559,E2 -8088.559} C_VEL
LIN {X 0,Y 460.695,Z 324.595,A -85,B 0,C 180,E1 -8092.108,E2 -8092.108} C_VEL
LIN {X 0,Y 460.694,Z 324.596,A -85,B 0,C 180,E1 -8094.748,E2 -8094.748} C_VEL
LIN {X 0,Y 460.823,Z 324.585,A -85,B 0,C 180,E1 -8097.377,E2 -8097.377} C_VEL
LIN {X 0,Y 460.852,Z 324.575,A -85,B 0,C 180,E1 -8100,E2 -8100} C_VEL
LIN {X 0,Y 460.824,Z 324.58,A -85,B 0,C 180,E1 -8102.622,E2 -8102.622} C_VEL
LIN {X 0,Y 460.7,Z 324.594,A -85,B 0,C 180,E1 -8106.13,E2 -8106.13} C_VEL
LIN {X 0,Y 460.627,Z 324.608,A -85,B 0,C 180,E1 -8108.776,E2 -8108.776} C_VEL
LIN {X 0,Y 460.612,Z 324.607,A -85,B 0,C 180,E1 -8112.444,E2 -8112.444} C_VEL
LIN {X 0,Y 460.598,Z 324.607,A -85,B 0,C 180,E1 -8115.997,E2 -8115.997} C_VEL
LIN {X 0,Y 460.569,Z 324.616,A -85,B 0,C 180,E1 -8118.902,E2 -8118.902} C_VEL
LIN {X 0,Y 460.513,Z 324.617,A -85,B 0,C 180,E1 -8121.485,E2 -8121.485} C_VEL
LIN {X 0,Y 460.539,Z 324.618,A -85,B 0,C 180,E1 -8124.332,E2 -8124.332} C_VEL
LIN {X 0,Y 460.57,Z 324.611,A -85,B 0,C 180,E1 -8127.243,E2 -8127.243} C_VEL
LIN {X 0,Y 460.508,Z 324.623,A -85,B 0,C 180,E1 -8130.24,E2 -8130.24} C_VEL
LIN {X 0,Y 460.526,Z 324.615,A -85,B 0,C 180,E1 -8133.324,E2 -8133.324} C_VEL
LIN {X 0,Y 460.475,Z 324.627,A -85,B 0,C 180,E1 -8136.529,E2 -8136.529} C_VEL
LIN {X 0,Y 460.571,Z 324.613,A -85,B 0,C 180,E1 -8139.858,E2 -8139.858} C_VEL
LIN {X 0,Y 460.539,Z 324.614,A -85,B 0,C 180,E1 -8142.904,E2 -8142.904} C_VEL
LIN {X 0,Y 460.508,Z 324.622,A -85,B 0,C 180,E1 -8145.83,E2 -8145.83} C_VEL
LIN {X 0,Y 460.535,Z 324.614,A -85,B 0,C 180,E1 -8148.989,E2 -8148.989} C_VEL
LIN {X 0,Y 460.536,Z 324.615,A -85,B 0,C 180,E1 -8151.268,E2 -8151.268} C_VEL
LIN {X 0,Y 460.509,Z 324.618,A -85,B 0,C 180,E1 -8154.554,E2 -8154.554} C_VEL
LIN {X 0,Y 460.529,Z 324.622,A -85,B 0,C 180,E1 -8157.716,E2 -8157.716} C_VEL
LIN {X 0,Y 460.536,Z 324.614,A -85,B 0,C 180,E1 -8160.769,E2 -8160.769} C_VEL
LIN {X 0,Y 460.565,Z 324.617,A -85,B 0,C 180,E1 -8163.735,E2 -8163.735} C_VEL
LIN {X 0,Y 460.542,Z 324.613,A -85,B 0,C 180,E1 -8166.624,E2 -8166.624} C_VEL
LIN {X 0,Y 460.549,Z 324.62,A -85,B 0,C 180,E1 -8169.453,E2 -8169.453} C_VEL
LIN {X 0,Y 460.556,Z 324.615,A -85,B 0,C 180,E1 -8172.23,E2 -8172.23} C_VEL
LIN {X 0,Y 460.564,Z 324.617,A -85,B 0,C 180,E1 -8174.965,E2 -8174.965} C_VEL
LIN {X 0,Y 460.608,Z 324.608,A -85,B 0,C 180,E1 -8178.559,E2 -8178.559} C_VEL
LIN {X 0,Y 460.574,Z 324.614,A -85,B 0,C 180,E1 -8179.211,E2 -8179.211} C_VEL
LIN {X 0,Y 459.919,Z 324.7,A -85,B 0,C 180,E1 -8179.941,E2 -8179.941} C_VEL
LIN {X 0,Y 457.102,Z 325.055,A -85,B 0,C 180,E1 -8181.128,E2 -8181.128} C_VEL
LIN {X 0,Y 454.723,Z 325.349,A -85,B 0,C 180,E1 -8182.085,E2 -8182.085} C_VEL
LIN {X 0,Y 453.711,Z 325.472,A -85,B 0,C 180,E1 -8182.824,E2 -8182.824} C_VEL
LIN {X 0,Y 453.633,Z 325.479,A -85,B 0,C 180,E1 -8183.074,E2 -8183.074} C_VEL
LIN {X 0,Y 453.67,Z 325.474,A -85,B 0,C 180,E1 -8184.667,E2 -8184.667} C_VEL
LIN {X 0,Y 453.762,Z 325.465,A -85,B 0,C 180,E1 -8187.337,E2 -8187.337} C_VEL
LIN {X 0,Y 453.821,Z 325.455,A -85,B 0,C 180,E1 -8190,E2 -8190} C_VEL
LIN {X 0,Y 453.762,Z 325.465,A -85,B 0,C 180,E1 -8192.663,E2 -8192.663} C_VEL
LIN {X 0,Y 453.676,Z 325.474,A -85,B 0,C 180,E1 -8196.225,E2 -8196.225} C_VEL
LIN {X 0,Y 453.589,Z 325.486,A -85,B 0,C 180,E1 -8198.913,E2 -8198.913} C_VEL
LIN {X 0,Y 453.56,Z 325.489,A -85,B 0,C 180,E1 -8202.529,E2 -8202.529} C_VEL
LIN {X 0,Y 453.541,Z 325.491,A -85,B 0,C 180,E1 -8206.196,E2 -8206.196} C_VEL
LIN {X 0,Y 453.517,Z 325.493,A -85,B 0,C 180,E1 -8209.041,E2 -8209.041} C_VEL
LIN {X 0,Y 453.472,Z 325.495,A -85,B 0,C 180,E1 -8211.836,E2 -8211.836} C_VEL
LIN {X 0,Y 453.51,Z 325.493,A -85,B 0,C 180,E1 -8214.735,E2 -8214.735} C_VEL
LIN {X 0,Y 453.534,Z 325.49,A -85,B 0,C 180,E1 -8217.961,E2 -8217.961} C_VEL
LIN {X 0,Y 453.463,Z 325.496,A -85,B 0,C 180,E1 -8221.526,E2 -8221.526} C_VEL
LIN {X 0,Y 453.485,Z 325.494,A -85,B 0,C 180,E1 -8224.778,E2 -8224.778} C_VEL
LIN {X 0,Y 453.477,Z 325.498,A -85,B 0,C 180,E1 -8228.31,E2 -8228.31} C_VEL
LIN {X 0,Y 453.512,Z 325.491,A -85,B 0,C 180,E1 -8230.607,E2 -8230.607} C_VEL
LIN {X 0,Y 453.462,Z 325.499,A -85,B 0,C 180,E1 -8234.221,E2 -8234.221} C_VEL
LIN {X 0,Y 453.488,Z 325.492,A -85,B 0,C 180,E1 -8237.009,E2 -8237.009} C_VEL
LIN {X 0,Y 453.525,Z 325.488,A -85,B 0,C 180,E1 -8240.555,E2 -8240.555} C_VEL
LIN {X 0,Y 453.451,Z 325.502,A -85,B 0,C 180,E1 -8243.918,E2 -8243.918} C_VEL
LIN {X 0,Y 453.48,Z 325.495,A -85,B 0,C 180,E1 -8247.152,E2 -8247.152} C_VEL
LIN {X 0,Y 453.472,Z 325.495,A -85,B 0,C 180,E1 -8250.269,E2 -8250.269} C_VEL
LIN {X 0,Y 453.504,Z 325.496,A -85,B 0,C 180,E1 -8253.294,E2 -8253.294} C_VEL
LIN {X 0,Y 453.5,Z 325.491,A -85,B 0,C 180,E1 -8256.239,E2 -8256.239} C_VEL
LIN {X 0,Y 453.481,Z 325.498,A -85,B 0,C 180,E1 -8259.118,E2 -8259.118} C_VEL
LIN {X 0,Y 453.509,Z 325.49,A -85,B 0,C 180,E1 -8261.945,E2 -8261.945} C_VEL
LIN {X 0,Y 453.538,Z 325.488,A -85,B 0,C 180,E1 -8264.727,E2 -8264.727} C_VEL
LIN {X 0,Y 453.558,Z 325.484,A -85,B 0,C 180,E1 -8268.379,E2 -8268.379} C_VEL
LIN {X 0,Y 453.651,Z 325.472,A -85,B 0,C 180,E1 -8271.986,E2 -8271.986} C_VEL
LIN {X 0,Y 453.666,Z 325.474,A -85,B 0,C 180,E1 -8274.667,E2 -8274.667} C_VEL
LIN {X 0,Y 453.764,Z 325.46,A -85,B 0,C 180,E1 -8277.337,E2 -8277.337} C_VEL
LIN {X 0,Y 453.822,Z 325.451,A -85,B 0,C 180,E1 -8280,E2 -8280} C_VEL
LIN {X 0,Y 453.764,Z 325.465,A -85,B 0,C 180,E1 -8282.664,E2 -8282.664} C_VEL
LIN {X 0,Y 453.669,Z 325.472,A -85,B 0,C 180,E1 -8286.226,E2 -8286.226} C_VEL
LIN {X 0,Y 453.592,Z 325.483,A -85,B 0,C 180,E1 -8288.914,E2 -8288.914} C_VEL
LIN {X 0,Y 453.563,Z 325.491,A -85,B 0,C 180,E1 -8292.529,E2 -8292.529} C_VEL
LIN {X 0,Y 453.544,Z 325.49,A -85,B 0,C 180,E1 -8296.196,E2 -8296.196} C_VEL
LIN {X 0,Y 453.517,Z 325.489,A -85,B 0,C 180,E1 -8299.04,E2 -8299.04} C_VEL
LIN {X 0,Y 453.477,Z 325.496,A -85,B 0,C 180,E1 -8301.837,E2 -8301.837} C_VEL
LIN {X 0,Y 453.501,Z 325.492,A -85,B 0,C 180,E1 -8304.736,E2 -8304.736} C_VEL
LIN {X 0,Y 453.533,Z 325.492,A -85,B 0,C 180,E1 -8307.96,E2 -8307.96} C_VEL
LIN {X 0,Y 453.466,Z 325.497,A -85,B 0,C 180,E1 -8311.526,E2 -8311.526} C_VEL
LIN {X 0,Y 453.488,Z 325.493,A -85,B 0,C 180,E1 -8314.778,E2 -8314.778} C_VEL
LIN {X 0,Y 453.466,Z 325.502,A -85,B 0,C 180,E1 -8318.312,E2 -8318.312} C_VEL
LIN {X 0,Y 453.495,Z 325.498,A -85,B 0,C 180,E1 -8320.609,E2 -8320.609} C_VEL
LIN {X 0,Y 453.609,Z 326.318,A -85,B 0,C 180,E1 -8321.954,E2 -8321.954} C_VEL
LIN {X 0,Y 454.151,Z 330.123,A -85,B 0,C 180,E1 -8325.386,E2 -8325.386} C_VEL
LIN {X 0,Y 454.379,Z 333.221,A -85,B 0,C 180,E1 -8327.939,E2 -8327.939} C_VEL
LIN {X 0,Y 454.235,Z 336.834,A -85,B 0,C 180,E1 -8330.68,E2 -8330.68} C_VEL
LIN {X 0,Y 454.019,Z 340.937,A -85,B 0,C 180,E1 -8333.605,E2 -8333.605} C_VEL
LIN {X 0,Y 453.727,Z 345.656,A -85,B 0,C 180,E1 -8336.766,E2 -8336.766} C_VEL
LIN {X 0,Y 453.486,Z 349.519,A -85,B 0,C 180,E1 -8339.241,E2 -8339.241} C_VEL
LIN {X 0,Y 453.253,Z 354.471,A -85,B 0,C 180,E1 -8342.279,E2 -8342.279} C_VEL
LIN {X 0,Y 452.991,Z 359.491,A -85,B 0,C 180,E1 -8345.235,E2 -8345.235} C_VEL
LIN {X 0,Y 452.798,Z 365.468,A -85,B 0,C 180,E1 -8348.635,E2 -8348.635} C_VEL
LIN {X 0,Y 452.629,Z 371.406,A -85,B 0,C 180,E1 -8351.908,E2 -8351.908} C_VEL
LIN {X 0,Y 452.558,Z 375.588,A -85,B 0,C 180,E1 -8354.136,E2 -8354.136} C_VEL
LIN {X 0,Y 454.317,Z 385.328,A -85,B 0,C 180,E1 -8354.461,E2 -8354.461} C_VEL
LIN {X 0,Y 455.651,Z 394.616,A -85,B 0,C 180,E1 -8354.856,E2 -8354.856} C_VEL
LIN {X 0,Y 456.112,Z 399.784,A -85,B 0,C 180,E1 -8355.1,E2 -8355.1} C_VEL
LIN {X 0,Y 455.511,Z 412.502,A -85,B 0,C 180,E1 -8355.822,E2 -8355.822} C_VEL
LIN {X 0,Y 455.025,Z 421.781,A -85,B 0,C 180,E1 -8356.49,E2 -8356.49} C_VEL
LIN {X 0,Y 454.62,Z 430.223,A -85,B 0,C 180,E1 -8357.223,E2 -8357.223} C_VEL
LIN {X 0,Y 454.153,Z 439.263,A -85,B 0,C 180,E1 -8358.168,E2 -8358.168} C_VEL
LIN {X 0,Y 453.721,Z 446.483,A -85,B 0,C 180,E1 -8359.062,E2 -8359.062} C_VEL
LIN {X 0,Y 453.434,Z 452.688,A -85,B 0,C 180,E1 -8359.958,E2 -8359.958} C_VEL
LIN {X 0,Y 453.104,Z 459.226,A -85,B 0,C 180,E1 -8361.077,E2 -8361.077} C_VEL
LIN {X 0,Y 452.893,Z 463.727,A -85,B 0,C 180,E1 -8361.972,E2 -8361.972} C_VEL
LIN {X 0,Y 452.648,Z 469.372,A -85,B 0,C 180,E1 -8363.358,E2 -8363.358} C_VEL
LIN {X 0,Y 452.57,Z 473.541,A -85,B 0,C 180,E1 -8364.654,E2 -8364.654} C_VEL
LIN {X 0,Y 452.489,Z 475.905,A -85,B 0,C 180,E1 -8365.546,E2 -8365.546} C_VEL
LIN {X 0,Y 452.481,Z 477.702,A -85,B 0,C 180,E1 -8366.438,E2 -8366.438} C_VEL
LIN {X 0,Y 452.437,Z 480.143,A -85,B 0,C 180,E1 -8368.22,E2 -8368.22} C_VEL
LIN {X 0,Y 452.429,Z 480.73,A -85,B 0,C 180,E1 -8369.11,E2 -8369.11} C_VEL
LIN {X 0,Y 452.429,Z 480.73,A -85,B 0,C 180,E1 -8370.89,E2 -8370.89} C_VEL
LIN {X 0,Y 452.437,Z 480.143,A -85,B 0,C 180,E1 -8371.78,E2 -8371.78} C_VEL
LIN {X 0,Y 452.481,Z 477.702,A -85,B 0,C 180,E1 -8373.562,E2 -8373.562} C_VEL
LIN {X 0,Y 452.55,Z 474.757,A -85,B 0,C 180,E1 -8374.9,E2 -8374.9} C_VEL
LIN {X 0,Y 452.605,Z 470.77,A -85,B 0,C 180,E1 -8376.24,E2 -8376.24} C_VEL
LIN {X 0,Y 452.814,Z 465.643,A -85,B 0,C 180,E1 -8377.581,E2 -8377.581} C_VEL
LIN {X 0,Y 453.052,Z 460.382,A -85,B 0,C 180,E1 -8378.699,E2 -8378.699} C_VEL
LIN {X 0,Y 453.344,Z 454.064,A -85,B 0,C 180,E1 -8379.818,E2 -8379.818} C_VEL
LIN {X 0,Y 453.618,Z 448.11,A -85,B 0,C 180,E1 -8380.715,E2 -8380.715} C_VEL
LIN {X 0,Y 454.044,Z 441.183,A -85,B 0,C 180,E1 -8381.608,E2 -8381.608} C_VEL
LIN {X 0,Y 454.475,Z 433,A -85,B 0,C 180,E1 -8382.503,E2 -8382.503} C_VEL
LIN {X 0,Y 454.846,Z 424.502,A -85,B 0,C 180,E1 -8383.286,E2 -8383.286} C_VEL
LIN {X 0,Y 455.31,Z 415.766,A -85,B 0,C 180,E1 -8383.956,E2 -8383.956} C_VEL
LIN {X 0,Y 455.766,Z 406.005,A -85,B 0,C 180,E1 -8384.569,E2 -8384.569} C_VEL
LIN {X 0,Y 456.135,Z 398.498,A -85,B 0,C 180,E1 -8384.956,E2 -8384.956} C_VEL
LIN {X 0,Y 454.6,Z 387.135,A -85,B 0,C 180,E1 -8385.47,E2 -8385.47} C_VEL
LIN {X 0,Y 452.714,Z 376.834,A -85,B 0,C 180,E1 -8385.832,E2 -8385.832} C_VEL
LIN {X 0,Y 452.556,Z 375.517,A -85,B 0,C 180,E1 -8385.896,E2 -8385.896} C_VEL
LIN {X 0,Y 452.679,Z 369.685,A -85,B 0,C 180,E1 -8389.028,E2 -8389.028} C_VEL
LIN {X 0,Y 452.799,Z 364.564,A -85,B 0,C 180,E1 -8391.87,E2 -8391.87} C_VEL
LIN {X 0,Y 452.989,Z 359.489,A -85,B 0,C 180,E1 -8394.765,E2 -8394.765} C_VEL
LIN {X 0,Y 453.253,Z 354.181,A -85,B 0,C 180,E1 -8397.892,E2 -8397.892} C_VEL
LIN {X 0,Y 453.492,Z 349.519,A -85,B 0,C 180,E1 -8400.758,E2 -8400.758} C_VEL
LIN {X 0,Y 453.762,Z 344.647,A -85,B 0,C 180,E1 -8403.888,E2 -8403.888} C_VEL
LIN {X 0,Y 454.02,Z 339.874,A -85,B 0,C 180,E1 -8407.135,E2 -8407.135} C_VEL
LIN {X 0,Y 454.194,Z 336.729,A -85,B 0,C 180,E1 -8409.376,E2 -8409.376} C_VEL
LIN {X 0,Y 454.377,Z 333.196,A -85,B 0,C 180,E1 -8412.06,E2 -8412.06} C_VEL
LIN {X 0,Y 454.146,Z 330.111,A -85,B 0,C 180,E1 -8414.613,E2 -8414.613} C_VEL
LIN {X 0,Y 453.567,Z 326.138,A -85,B 0,C 180,E1 -8418.219,E2 -8418.219} C_VEL
LIN {X 0,Y 453.496,Z 325.497,A -85,B 0,C 180,E1 -8419.409,E2 -8419.409} C_VEL
LIN {X 0,Y 453.451,Z 325.505,A -85,B 0,C 180,E1 -8422.227,E2 -8422.227} C_VEL
LIN {X 0,Y 453.488,Z 325.497,A -85,B 0,C 180,E1 -8425.222,E2 -8425.222} C_VEL
LIN {X 0,Y 453.466,Z 325.497,A -85,B 0,C 180,E1 -8428.474,E2 -8428.474} C_VEL
LIN {X 0,Y 453.533,Z 325.492,A -85,B 0,C 180,E1 -8432.04,E2 -8432.04} C_VEL
LIN {X 0,Y 453.501,Z 325.492,A -85,B 0,C 180,E1 -8435.264,E2 -8435.264} C_VEL
LIN {X 0,Y 453.48,Z 325.494,A -85,B 0,C 180,E1 -8438.415,E2 -8438.415} C_VEL
LIN {X 0,Y 453.522,Z 325.489,A -85,B 0,C 180,E1 -8441.008,E2 -8441.008} C_VEL
LIN {X 0,Y 453.569,Z 325.486,A -85,B 0,C 180,E1 -8443.879,E2 -8443.879} C_VEL
LIN {X 0,Y 453.563,Z 325.491,A -85,B 0,C 180,E1 -8447.471,E2 -8447.471} C_VEL
LIN {X 0,Y 453.592,Z 325.483,A -85,B 0,C 180,E1 -8451.086,E2 -8451.086} C_VEL
LIN {X 0,Y 453.669,Z 325.472,A -85,B 0,C 180,E1 -8453.774,E2 -8453.774} C_VEL
LIN {X 0,Y 453.764,Z 325.465,A -85,B 0,C 180,E1 -8457.336,E2 -8457.336} C_VEL
LIN {X 0,Y 453.822,Z 325.451,A -85,B 0,C 180,E1 -8460,E2 -8460} C_VEL
LIN {X 0,Y 453.764,Z 325.46,A -85,B 0,C 180,E1 -8462.663,E2 -8462.663} C_VEL
LIN {X 0,Y 453.668,Z 325.47,A -85,B 0,C 180,E1 -8466.225,E2 -8466.225} C_VEL
LIN {X 0,Y 453.591,Z 325.487,A -85,B 0,C 180,E1 -8468.913,E2 -8468.913} C_VEL
LIN {X 0,Y 453.562,Z 325.486,A -85,B 0,C 180,E1 -8472.528,E2 -8472.528} C_VEL
LIN {X 0,Y 453.543,Z 325.487,A -85,B 0,C 180,E1 -8476.195,E2 -8476.195} C_VEL
LIN {X 0,Y 453.518,Z 325.492,A -85,B 0,C 180,E1 -8479.04,E2 -8479.04} C_VEL
LIN {X 0,Y 453.474,Z 325.494,A -85,B 0,C 180,E1 -8481.836,E2 -8481.836} C_VEL
LIN {X 0,Y 453.511,Z 325.495,A -85,B 0,C 180,E1 -8484.734,E2 -8484.734} C_VEL
LIN {X 0,Y 453.529,Z 325.489,A -85,B 0,C 180,E1 -8487.959,E2 -8487.959} C_VEL
LIN {X 0,Y 453.464,Z 325.495,A -85,B 0,C 180,E1 -8491.525,E2 -8491.525} C_VEL
LIN {X 0,Y 453.486,Z 325.495,A -85,B 0,C 180,E1 -8494.777,E2 -8494.777} C_VEL
LIN {X 0,Y 453.478,Z 325.501,A -85,B 0,C 180,E1 -8498.31,E2 -8498.31} C_VEL
LIN {X 0,Y 453.513,Z 325.492,A -85,B 0,C 180,E1 -8500.606,E2 -8500.606} C_VEL
LIN {X 0,Y 453.478,Z 325.493,A -85,B 0,C 180,E1 -8503.247,E2 -8503.247} C_VEL
LIN {X 0,Y 453.462,Z 325.499,A -85,B 0,C 180,E1 -8505.779,E2 -8505.779} C_VEL
LIN {X 0,Y 453.512,Z 325.491,A -85,B 0,C 180,E1 -8509.405,E2 -8509.405} C_VEL
LIN {X 0,Y 453.472,Z 325.498,A -85,B 0,C 180,E1 -8512.223,E2 -8512.223} C_VEL
LIN {X 0,Y 453.485,Z 325.494,A -85,B 0,C 180,E1 -8515.222,E2 -8515.222} C_VEL
LIN {X 0,Y 453.463,Z 325.496,A -85,B 0,C 180,E1 -8518.474,E2 -8518.474} C_VEL
LIN {X 0,Y 453.534,Z 325.49,A -85,B 0,C 180,E1 -8522.039,E2 -8522.039} C_VEL
LIN {X 0,Y 453.51,Z 325.493,A -85,B 0,C 180,E1 -8525.265,E2 -8525.265} C_VEL
LIN {X 0,Y 453.476,Z 325.494,A -85,B 0,C 180,E1 -8528.415,E2 -8528.415} C_VEL
LIN {X 0,Y 453.519,Z 325.493,A -85,B 0,C 180,E1 -8531.009,E2 -8531.009} C_VEL
LIN {X 0,Y 453.565,Z 325.488,A -85,B 0,C 180,E1 -8533.88,E2 -8533.88} C_VEL
LIN {X 0,Y 453.56,Z 325.489,A -85,B 0,C 180,E1 -8537.471,E2 -8537.471} C_VEL
LIN {X 0,Y 453.589,Z 325.486,A -85,B 0,C 180,E1 -8541.087,E2 -8541.087} C_VEL
LIN {X 0,Y 453.633,Z 325.479,A -85,B 0,C 180,E1 -8543.074,E2 -8543.074} C_VEL
LIN {X 0,Y 452.948,Z 325.565,A -85,B 0,C 180,E1 -8543.815,E2 -8543.815} C_VEL
LIN {X 0,Y 449.998,Z 325.935,A -85,B 0,C 180,E1 -8545.016,E2 -8545.016} C_VEL
LIN {X 0,Y 447.574,Z 326.234,A -85,B 0,C 180,E1 -8545.986,E2 -8545.986} C_VEL
LIN {X 0,Y 446.636,Z 326.352,A -85,B 0,C 180,E1 -8546.736,E2 -8546.736} C_VEL
LIN {X 0,Y 446.616,Z 326.353,A -85,B 0,C 180,E1 -8546.99,E2 -8546.99} C_VEL
LIN {X 0,Y 446.791,Z 326.331,A -85,B 0,C 180,E1 -8550,E2 -8550} C_VEL
LIN {X 0,Y 446.706,Z 326.344,A -85,B 0,C 180,E1 -8552.705,E2 -8552.705} C_VEL
LIN {X 0,Y 446.645,Z 326.35,A -85,B 0,C 180,E1 -8556.324,E2 -8556.324} C_VEL
LIN {X 0,Y 446.535,Z 326.364,A -85,B 0,C 180,E1 -8559.055,E2 -8559.055} C_VEL
LIN {X 0,Y 446.518,Z 326.368,A -85,B 0,C 180,E1 -8562.73,E2 -8562.73} C_VEL
LIN {X 0,Y 446.492,Z 326.369,A -85,B 0,C 180,E1 -8566.228,E2 -8566.228} C_VEL
LIN {X 0,Y 446.466,Z 326.368,A -85,B 0,C 180,E1 -8569.303,E2 -8569.303} C_VEL
LIN {X 0,Y 446.415,Z 326.378,A -85,B 0,C 180,E1 -8572.2,E2 -8572.2} C_VEL
LIN {X 0,Y 446.454,Z 326.369,A -85,B 0,C 180,E1 -8575.152,E2 -8575.152} C_VEL
LIN {X 0,Y 446.481,Z 326.371,A -85,B 0,C 180,E1 -8578.179,E2 -8578.179} C_VEL
LIN {X 0,Y 446.416,Z 326.375,A -85,B 0,C 180,E1 -8581.775,E2 -8581.775} C_VEL
LIN {X 0,Y 446.427,Z 326.375,A -85,B 0,C 180,E1 -8584.523,E2 -8584.523} C_VEL
LIN {X 0,Y 446.432,Z 326.379,A -85,B 0,C 180,E1 -8588.083,E2 -8588.083} C_VEL
LIN {X 0,Y 446.439,Z 326.37,A -85,B 0,C 180,E1 -8590.92,E2 -8590.92} C_VEL
LIN {X 0,Y 446.413,Z 326.38,A -85,B 0,C 180,E1 -8593.844,E2 -8593.844} C_VEL
LIN {X 0,Y 446.443,Z 326.372,A -85,B 0,C 180,E1 -8596.397,E2 -8596.397} C_VEL
LIN {X 0,Y 446.464,Z 326.375,A -85,B 0,C 180,E1 -8599.805,E2 -8599.805} C_VEL
LIN {X 0,Y 446.428,Z 326.375,A -85,B 0,C 180,E1 -8602.124,E2 -8602.124} C_VEL
LIN {X 0,Y 446.426,Z 326.377,A -85,B 0,C 180,E1 -8605.477,E2 -8605.477} C_VEL
LIN {X 0,Y 446.413,Z 326.374,A -85,B 0,C 180,E1 -8608.7,E2 -8608.7} C_VEL
LIN {X 0,Y 446.482,Z 326.369,A -85,B 0,C 180,E1 -8611.822,E2 -8611.822} C_VEL
LIN {X 0,Y 446.454,Z 326.37,A -85,B 0,C 180,E1 -8614.848,E2 -8614.848} C_VEL
LIN {X 0,Y 446.446,Z 326.37,A -85,B 0,C 180,E1 -8618.246,E2 -8618.246} C_VEL
LIN {X 0,Y 446.455,Z 326.371,A -85,B 0,C 180,E1 -8621.65,E2 -8621.65} C_VEL
LIN {X 0,Y 446.506,Z 326.363,A -85,B 0,C 180,E1 -8624.48,E2 -8624.48} C_VEL
LIN {X 0,Y 446.516,Z 326.361,A -85,B 0,C 180,E1 -8628.194,E2 -8628.194} C_VEL
LIN {X 0,Y 446.599,Z 326.351,A -85,B 0,C 180,E1 -8631.858,E2 -8631.858} C_VEL
LIN {X 0,Y 446.641,Z 326.348,A -85,B 0,C 180,E1 -8634.583,E2 -8634.583} C_VEL
LIN {X 0,Y 446.708,Z 326.34,A -85,B 0,C 180,E1 -8637.295,E2 -8637.295} C_VEL
LIN {X 0,Y 446.792,Z 326.327,A -85,B 0,C 180,E1 -8640,E2 -8640} C_VEL
LIN {X 0,Y 446.707,Z 326.344,A -85,B 0,C 180,E1 -8642.706,E2 -8642.706} C_VEL
LIN {X 0,Y 446.639,Z 326.349,A -85,B 0,C 180,E1 -8646.324,E2 -8646.324} C_VEL
LIN {X 0,Y 446.538,Z 326.36,A -85,B 0,C 180,E1 -8649.056,E2 -8649.056} C_VEL
LIN {X 0,Y 446.521,Z 326.365,A -85,B 0,C 180,E1 -8652.73,E2 -8652.73} C_VEL
LIN {X 0,Y 446.496,Z 326.368,A -85,B 0,C 180,E1 -8656.228,E2 -8656.228} C_VEL
LIN {X 0,Y 446.468,Z 326.367,A -85,B 0,C 180,E1 -8659.304,E2 -8659.304} C_VEL
LIN {X 0,Y 446.419,Z 326.38,A -85,B 0,C 180,E1 -8662.2,E2 -8662.2} C_VEL
